LIN {X 0.031,Y -492.677,Z 365.442,A 0.000,B 0.000,C 90.000,E1 115.591} C_DIS
LIN {X -0.098,Y -489.173,Z 365.437,A 0.000,B 0.000,C 90.000,E1 114.695} C_DIS
LIN {X -0.238,Y -484.944,Z 365.431,A 0.000,B 0.000,C 90.000,E1 113.643} C_DIS
LIN {X 0.196,Y -479.146,Z 365.424,A 0.000,B 0.000,C 90.000,E1 112.206} C_DIS
LIN {X -0.106,Y -472.835,Z 365.416,A 0.000,B 0.000,C 90.000,E1 110.844} C_DIS
LIN {X -0.106,Y -464.087,Z 365.405,A 0.000,B 0.000,C 90.000,E1 108.960} C_DIS
LIN {X -0.172,Y -460.381,Z 365.401,A 0.000,B 0.000,C 90.000,E1 108.181} C_DIS
LIN {X -0.212,Y -460.379,Z 365.401,A 0.000,B 0.000,C 90.000,E1 108.181} C_DIS
LIN {X 0.188,Y -467.863,Z 365.383,A 0.000,B 0.000,C 90.000,E1 104.828} C_DIS
LIN {X -0.251,Y -475.421,Z 365.358,A 0.000,B 0.000,C 90.000,E1 100.489} C_DIS
LIN {X 0.054,Y -476.073,Z 365.356,A 0.000,B 0.000,C 90.000,E1 100.141} C_DIS
LIN {X -0.142,Y -481.996,Z 365.331,A 0.000,B 0.000,C 90.000,E1 95.511} C_DIS
LIN {X -0.161,Y -482.512,Z 365.325,A 0.000,B 0.000,C 90.000,E1 94.588} C_DIS
LIN {X 0.129,Y -485.445,Z 365.305,A 0.000,B 0.000,C 90.000,E1 90.859} C_DIS
LIN {X -0.219,Y -485.505,Z 365.301,A 0.000,B 0.000,C 90.000,E1 90.286} C_DIS
LIN {X 0.162,Y -486.380,Z 365.281,A 0.000,B 0.000,C 90.000,E1 86.560} C_DIS
LIN {X -0.014,Y -486.365,Z 365.279,A 0.000,B 0.000,C 90.000,E1 86.274} C_DIS
LIN {X 0.075,Y -484.690,Z 365.254,A 0.000,B 0.000,C 90.000,E1 81.659} C_DIS
LIN {X 0.220,Y -484.078,Z 365.250,A 0.000,B 0.000,C 90.000,E1 81.027} C_DIS
LIN {X -0.123,Y -480.642,Z 365.228,A 0.000,B 0.000,C 90.000,E1 77.061} C_DIS
LIN {X -0.158,Y -480.354,Z 365.226,A 0.000,B 0.000,C 90.000,E1 76.756} C_DIS
LIN {X -0.155,Y -475.588,Z 365.208,A 0.000,B 0.000,C 90.000,E1 73.433} C_DIS
LIN {X 0.260,Y -475.616,Z 365.208,A 0.000,B 0.000,C 90.000,E1 73.378} C_DIS
LIN {X 0.037,Y -482.998,Z 365.201,A 0.000,B 0.000,C 90.000,E1 72.236} C_DIS
LIN {X -0.116,Y -486.733,Z 365.198,A 0.000,B 0.000,C 90.000,E1 71.638} C_DIS
LIN {X -0.244,Y -490.378,Z 365.195,A 0.000,B 0.000,C 90.000,E1 71.040} C_DIS
LIN {X 0.028,Y -493.043,Z 365.192,A 0.000,B 0.000,C 90.000,E1 70.550} C_DIS
LIN {X -0.145,Y -495.741,Z 365.189,A 0.000,B 0.000,C 90.000,E1 70.115} C_DIS
LIN {X 0.049,Y -499.772,Z 365.185,A 0.000,B 0.000,C 90.000,E1 69.337} C_DIS
LIN {X -0.208,Y -504.048,Z 365.180,A 0.000,B 0.000,C 90.000,E1 68.465} C_DIS
LIN {X -0.037,Y -506.775,Z 365.177,A 0.000,B 0.000,C 90.000,E1 67.847} C_DIS
LIN {X -0.105,Y -511.591,Z 365.170,A 0.000,B 0.000,C 90.000,E1 66.666} C_DIS
LIN {X -0.233,Y -514.726,Z 365.165,A 0.000,B 0.000,C 90.000,E1 65.793} C_DIS
LIN {X -0.114,Y -517.640,Z 365.161,A 0.000,B 0.000,C 90.000,E1 64.897} C_DIS
LIN {X 0.151,Y -519.464,Z 365.157,A 0.000,B 0.000,C 90.000,E1 64.280} C_DIS
LIN {X -0.139,Y -522.117,Z 365.152,A 0.000,B 0.000,C 90.000,E1 63.435} C_DIS
LIN {X -0.160,Y -527.061,Z 365.143,A 0.000,B 0.000,C 90.000,E1 61.691} C_DIS
LIN {X -0.088,Y -531.857,Z 365.133,A 0.000,B 0.000,C 90.000,E1 59.950} C_DIS
LIN {X 0.001,Y -534.996,Z 365.127,A 0.000,B 0.000,C 90.000,E1 58.791} C_DIS
LIN {X -0.138,Y -538.016,Z 365.120,A 0.000,B 0.000,C 90.000,E1 57.661} C_DIS
LIN {X 0.085,Y -542.351,Z 365.111,A 0.000,B 0.000,C 90.000,E1 55.928} C_DIS
LIN {X -0.111,Y -545.003,Z 365.105,A 0.000,B 0.000,C 90.000,E1 54.815} C_DIS
LIN {X -0.317,Y -546.812,Z 365.100,A 0.000,B 0.000,C 90.000,E1 53.989} C_DIS
LIN {X -0.087,Y -549.488,Z 365.092,A 0.000,B 0.000,C 90.000,E1 52.557} C_DIS
LIN {X 0.073,Y -550.750,Z 365.087,A 0.000,B 0.000,C 90.000,E1 51.698} C_DIS
LIN {X -0.187,Y -551.579,Z 365.083,A 0.000,B 0.000,C 90.000,E1 50.884} C_DIS
LIN {X -0.083,Y -552.180,Z 365.078,A 0.000,B 0.000,C 90.000,E1 50.033} C_DIS
LIN {X 0.036,Y -552.398,Z 365.075,A 0.000,B 0.000,C 90.000,E1 49.461} C_DIS
LIN {X 0.156,Y -552.500,Z 365.070,A 0.000,B 0.000,C 90.000,E1 48.609} C_DIS
LIN {X -0.091,Y -552.312,Z 365.066,A 0.000,B 0.000,C 90.000,E1 47.796} C_DIS
LIN {X 0.025,Y -551.870,Z 365.061,A 0.000,B 0.000,C 90.000,E1 46.944} C_DIS
LIN {X -0.264,Y -551.137,Z 365.056,A 0.000,B 0.000,C 90.000,E1 46.134} C_DIS
LIN {X -0.135,Y -549.862,Z 365.050,A 0.000,B 0.000,C 90.000,E1 45.000} C_DIS
LIN {X 0.007,Y -548.109,Z 365.042,A 0.000,B 0.000,C 90.000,E1 43.581} C_DIS
LIN {X 0.142,Y -545.398,Z 365.031,A 0.000,B 0.000,C 90.000,E1 41.595} C_DIS
LIN {X -0.145,Y -543.179,Z 365.022,A 0.000,B 0.000,C 90.000,E1 39.930} C_DIS
LIN {X -0.045,Y -540.492,Z 365.011,A 0.000,B 0.000,C 90.000,E1 37.935} C_DIS
LIN {X 0.066,Y -538.243,Z 365.001,A 0.000,B 0.000,C 90.000,E1 36.217} C_DIS
LIN {X -0.188,Y -535.980,Z 364.992,A 0.000,B 0.000,C 90.000,E1 34.532} C_DIS
LIN {X -0.052,Y -533.823,Z 364.982,A 0.000,B 0.000,C 90.000,E1 32.801} C_DIS
LIN {X 0.215,Y -532.034,Z 364.974,A 0.000,B 0.000,C 90.000,E1 31.337} C_DIS
LIN {X 0.160,Y -530.007,Z 364.965,A 0.000,B 0.000,C 90.000,E1 29.617} C_DIS
LIN {X -0.247,Y -527.759,Z 364.953,A 0.000,B 0.000,C 90.000,E1 27.641} C_DIS
LIN {X -0.028,Y -525.601,Z 364.942,A 0.000,B 0.000,C 90.000,E1 25.591} C_DIS
LIN {X 0.221,Y -523.874,Z 364.933,A 0.000,B 0.000,C 90.000,E1 23.823} C_DIS
LIN {X 0.061,Y -522.555,Z 364.924,A 0.000,B 0.000,C 90.000,E1 22.386} C_DIS
LIN {X -0.048,Y -520.702,Z 364.911,A 0.000,B 0.000,C 90.000,E1 20.066} C_DIS
LIN {X 0.144,Y -519.352,Z 364.900,A 0.000,B 0.000,C 90.000,E1 18.000} C_DIS
LIN {X -0.114,Y -518.754,Z 364.894,A 0.000,B 0.000,C 90.000,E1 16.858} C_DIS
LIN {X 0.207,Y -517.916,Z 364.882,A 0.000,B 0.000,C 90.000,E1 14.773} C_DIS
LIN {X -0.176,Y -517.362,Z 364.866,A 0.000,B 0.000,C 90.000,E1 11.883} C_DIS
LIN {X 0.149,Y -517.388,Z 364.853,A 0.000,B 0.000,C 90.000,E1 9.500} C_DIS
LIN {X 0.125,Y -517.389,Z 364.850,A 0.000,B 0.000,C 90.000,E1 8.916} C_DIS
LIN {X 0.007,Y -517.728,Z 364.845,A 0.000,B 0.000,C 90.000,E1 8.049} C_DIS
LIN {X -0.060,Y -519.631,Z 364.822,A 0.000,B 0.000,C 90.000,E1 3.955} C_DIS
LIN {X -0.082,Y -522.363,Z 364.804,A 0.000,B 0.000,C 90.000,E1 0.745} C_DIS
LIN {X -0.091,Y -526.446,Z 364.786,A 0.000,B 0.000,C 90.000,E1 357.478} C_DIS
LIN {X -0.247,Y -529.588,Z 364.775,A 0.000,B 0.000,C 90.000,E1 355.469} C_DIS
LIN {X -0.228,Y -533.117,Z 364.764,A 0.000,B 0.000,C 90.000,E1 353.451} C_DIS
LIN {X -0.116,Y -537.025,Z 364.752,A 0.000,B 0.000,C 90.000,E1 351.432} C_DIS
LIN {X 0.126,Y -545.013,Z 364.733,A 0.000,B 0.000,C 90.000,E1 347.993} C_DIS
LIN {X -0.031,Y -551.141,Z 364.721,A 0.000,B 0.000,C 90.000,E1 345.755} C_DIS
LIN {X 0.001,Y -556.922,Z 364.710,A 0.000,B 0.000,C 90.000,E1 343.795} C_DIS
LIN {X -0.106,Y -561.147,Z 364.702,A 0.000,B 0.000,C 90.000,E1 342.417} C_DIS
LIN {X 0.178,Y -566.255,Z 364.693,A 0.000,B 0.000,C 90.000,E1 340.732} C_DIS
LIN {X -0.126,Y -570.563,Z 364.685,A 0.000,B 0.000,C 90.000,E1 339.390} C_DIS
LIN {X 0.217,Y -575.641,Z 364.676,A 0.000,B 0.000,C 90.000,E1 337.720} C_DIS
LIN {X 0.286,Y -579.970,Z 364.669,A 0.000,B 0.000,C 90.000,E1 336.357} C_DIS
LIN {X 0.160,Y -586.014,Z 364.658,A 0.000,B 0.000,C 90.000,E1 334.485} C_DIS
LIN {X 0.052,Y -593.076,Z 364.647,A 0.000,B 0.000,C 90.000,E1 332.359} C_DIS
LIN {X -0.047,Y -596.678,Z 364.641,A 0.000,B 0.000,C 90.000,E1 331.307} C_DIS
LIN {X -0.093,Y -600.308,Z 364.635,A 0.000,B 0.000,C 90.000,E1 330.255} C_DIS
LIN {X 0.083,Y -605.802,Z 364.626,A 0.000,B 0.000,C 90.000,E1 328.663} C_DIS
LIN {X -0.157,Y -611.211,Z 364.617,A 0.000,B 0.000,C 90.000,E1 327.120} C_DIS
LIN {X -0.170,Y -617.620,Z 364.607,A 0.000,B 0.000,C 90.000,E1 325.308} C_DIS
LIN {X -0.028,Y -624.176,Z 364.597,A 0.000,B 0.000,C 90.000,E1 323.497} C_DIS
LIN {X 0.306,Y -628.949,Z 364.590,A 0.000,B 0.000,C 90.000,E1 322.190} C_DIS
LIN {X 0.350,Y -637.363,Z 364.577,A 0.000,B 0.000,C 90.000,E1 319.908} C_DIS
LIN {X 0.021,Y -641.197,Z 364.572,A 0.000,B 0.000,C 90.000,E1 318.933} C_DIS
LIN {X 0.090,Y -645.615,Z 364.565,A 0.000,B 0.000,C 90.000,E1 317.676} C_DIS
LIN {X 0.050,Y -653.617,Z 364.553,A 0.000,B 0.000,C 90.000,E1 315.445} C_DIS
LIN {X 0.291,Y -658.944,Z 364.544,A 0.000,B 0.000,C 90.000,E1 313.947} C_DIS
LIN {X -0.290,Y -664.100,Z 364.536,A 0.000,B 0.000,C 90.000,E1 312.528} C_DIS
LIN {X 0.164,Y -667.540,Z 364.531,A 0.000,B 0.000,C 90.000,E1 311.515} C_DIS
LIN {X -0.210,Y -671.484,Z 364.524,A 0.000,B 0.000,C 90.000,E1 310.334} C_DIS
LIN {X -0.085,Y -675.435,Z 364.517,A 0.000,B 0.000,C 90.000,E1 309.116} C_DIS
LIN {X -0.350,Y -678.537,Z 364.512,A 0.000,B 0.000,C 90.000,E1 308.177} C_DIS
LIN {X 0.382,Y -681.266,Z 364.507,A 0.000,B 0.000,C 90.000,E1 307.156} C_DIS
LIN {X 0.191,Y -683.841,Z 364.501,A 0.000,B 0.000,C 90.000,E1 306.217} C_DIS
LIN {X -0.372,Y -686.227,Z 364.496,A 0.000,B 0.000,C 90.000,E1 305.311} C_DIS
LIN {X 0.050,Y -688.341,Z 364.491,A 0.000,B 0.000,C 90.000,E1 304.326} C_DIS
LIN {X -0.097,Y -689.746,Z 364.487,A 0.000,B 0.000,C 90.000,E1 303.627} C_DIS
LIN {X 0.344,Y -690.890,Z 364.483,A 0.000,B 0.000,C 90.000,E1 302.880} C_DIS
LIN {X 0.074,Y -692.274,Z 364.478,A 0.000,B 0.000,C 90.000,E1 301.957} C_DIS
LIN {X 0.312,Y -692.953,Z 364.475,A 0.000,B 0.000,C 90.000,E1 301.465} C_DIS
LIN {X -0.165,Y -693.622,Z 364.471,A 0.000,B 0.000,C 90.000,E1 300.797} C_DIS
LIN {X -0.280,Y -693.986,Z 364.468,A 0.000,B 0.000,C 90.000,E1 300.335} C_DIS
LIN {X 0.101,Y -694.209,Z 364.463,A 0.000,B 0.000,C 90.000,E1 299.361} C_DIS
LIN {X -0.006,Y -694.162,Z 364.461,A 0.000,B 0.000,C 90.000,E1 298.899} C_DIS
LIN {X 0.134,Y -693.618,Z 364.457,A 0.000,B 0.000,C 90.000,E1 298.180} C_DIS
LIN {X 0.145,Y -692.090,Z 364.450,A 0.000,B 0.000,C 90.000,E1 297.001} C_DIS
LIN {X 0.189,Y -690.657,Z 364.445,A 0.000,B 0.000,C 90.000,E1 296.052} C_DIS
LIN {X 0.280,Y -689.460,Z 364.441,A 0.000,B 0.000,C 90.000,E1 295.335} C_DIS
LIN {X 0.288,Y -687.540,Z 364.436,A 0.000,B 0.000,C 90.000,E1 294.387} C_DIS
LIN {X 0.213,Y -684.989,Z 364.429,A 0.000,B 0.000,C 90.000,E1 293.206} C_DIS
LIN {X -0.103,Y -682.772,Z 364.424,A 0.000,B 0.000,C 90.000,E1 292.280} C_DIS
LIN {X -0.064,Y -679.228,Z 364.416,A 0.000,B 0.000,C 90.000,E1 290.844} C_DIS
LIN {X 0.055,Y -675.760,Z 364.408,A 0.000,B 0.000,C 90.000,E1 289.396} C_DIS
LIN {X 0.249,Y -673.445,Z 364.402,A 0.000,B 0.000,C 90.000,E1 288.417} C_DIS
LIN {X 0.112,Y -668.889,Z 364.392,A 0.000,B 0.000,C 90.000,E1 286.496} C_DIS
LIN {X 0.147,Y -663.586,Z 364.378,A 0.000,B 0.000,C 90.000,E1 284.064} C_DIS
LIN {X 0.152,Y -658.265,Z 364.362,A 0.000,B 0.000,C 90.000,E1 281.130} C_DIS
LIN {X 0.060,Y -654.842,Z 364.348,A 0.000,B 0.000,C 90.000,E1 278.681} C_DIS
LIN {X -0.150,Y -651.967,Z 364.332,A 0.000,B 0.000,C 90.000,E1 275.739} C_DIS
LIN {X 0.288,Y -650.524,Z 364.317,A 0.000,B 0.000,C 90.000,E1 272.980} C_DIS
LIN {X -0.294,Y -649.937,Z 364.304,A 0.000,B 0.000,C 90.000,E1 270.802} C_DIS
LIN {X 0.015,Y -650.410,Z 364.285,A 0.000,B 0.000,C 90.000,E1 267.306} C_DIS
LIN {X 0.112,Y -651.031,Z 364.277,A 0.000,B 0.000,C 90.000,E1 265.812} C_DIS
LIN {X 0.007,Y -651.804,Z 364.267,A 0.000,B 0.000,C 90.000,E1 264.090} C_DIS
LIN {X -0.180,Y -652.598,Z 364.256,A 0.000,B 0.000,C 90.000,E1 262.129} C_DIS
LIN {X -0.039,Y -652.961,Z 364.252,A 0.000,B 0.000,C 90.000,E1 261.376} C_DIS
LIN {X 0.105,Y -652.989,Z 364.248,A 0.000,B 0.000,C 90.000,E1 260.622} C_DIS
LIN {X -0.134,Y -652.869,Z 364.240,A 0.000,B 0.000,C 90.000,E1 259.162} C_DIS
LIN {X 0.268,Y -652.672,Z 364.232,A 0.000,B 0.000,C 90.000,E1 257.645} C_DIS
LIN {X -0.101,Y -652.414,Z 364.227,A 0.000,B 0.000,C 90.000,E1 256.937} C_DIS
LIN {X -0.085,Y -651.414,Z 364.221,A 0.000,B 0.000,C 90.000,E1 255.700} C_DIS
LIN {X 0.165,Y -650.736,Z 364.216,A 0.000,B 0.000,C 90.000,E1 254.936} C_DIS
LIN {X -0.050,Y -649.669,Z 364.212,A 0.000,B 0.000,C 90.000,E1 254.212} C_DIS
LIN {X 0.172,Y -648.378,Z 364.208,A 0.000,B 0.000,C 90.000,E1 253.449} C_DIS
LIN {X 0.083,Y -647.443,Z 364.205,A 0.000,B 0.000,C 90.000,E1 252.960} C_DIS
LIN {X -0.150,Y -645.773,Z 364.201,A 0.000,B 0.000,C 90.000,E1 252.236} C_DIS
LIN {X 0.214,Y -643.871,Z 364.197,A 0.000,B 0.000,C 90.000,E1 251.456} C_DIS
LIN {X 0.107,Y -642.470,Z 364.194,A 0.000,B 0.000,C 90.000,E1 250.967} C_DIS
LIN {X -0.345,Y -639.212,Z 364.189,A 0.000,B 0.000,C 90.000,E1 250.007} C_DIS
LIN {X 0.197,Y -635.669,Z 364.183,A 0.000,B 0.000,C 90.000,E1 248.954} C_DIS
LIN {X -0.128,Y -631.902,Z 364.178,A 0.000,B 0.000,C 90.000,E1 247.975} C_DIS
LIN {X 0.335,Y -626.967,Z 364.171,A 0.000,B 0.000,C 90.000,E1 246.666} C_DIS
LIN {X 0.140,Y -621.804,Z 364.164,A 0.000,B 0.000,C 90.000,E1 245.409} C_DIS
LIN {X -0.156,Y -615.473,Z 364.155,A 0.000,B 0.000,C 90.000,E1 243.896} C_DIS
LIN {X -0.352,Y -608.026,Z 364.145,A 0.000,B 0.000,C 90.000,E1 242.103} C_DIS
LIN {X -0.084,Y -601.654,Z 364.136,A 0.000,B 0.000,C 90.000,E1 240.511} C_DIS
LIN {X 0.063,Y -595.379,Z 364.127,A 0.000,B 0.000,C 90.000,E1 238.918} C_DIS
LIN {X -0.290,Y -585.515,Z 364.113,A 0.000,B 0.000,C 90.000,E1 236.294} C_DIS
LIN {X 0.159,Y -577.276,Z 364.099,A 0.000,B 0.000,C 90.000,E1 233.829} C_DIS
LIN {X 0.126,Y -572.773,Z 364.092,A 0.000,B 0.000,C 90.000,E1 232.477} C_DIS
LIN {X -0.316,Y -566.944,Z 364.083,A 0.000,B 0.000,C 90.000,E1 230.884} C_DIS
LIN {X 0.059,Y -558.457,Z 364.069,A 0.000,B 0.000,C 90.000,E1 228.366} C_DIS
LIN {X 0.317,Y -554.841,Z 364.063,A 0.000,B 0.000,C 90.000,E1 227.229} C_DIS
LIN {X -0.243,Y -550.314,Z 364.055,A 0.000,B 0.000,C 90.000,E1 225.891} C_DIS
LIN {X -0.130,Y -546.711,Z 364.049,A 0.000,B 0.000,C 90.000,E1 224.757} C_DIS
LIN {X -0.052,Y -540.419,Z 364.038,A 0.000,B 0.000,C 90.000,E1 222.771} C_DIS
LIN {X -0.098,Y -536.030,Z 364.030,A 0.000,B 0.000,C 90.000,E1 221.353} C_DIS
LIN {X -0.202,Y -529.943,Z 364.019,A 0.000,B 0.000,C 90.000,E1 219.358} C_DIS
LIN {X -0.002,Y -524.922,Z 364.009,A 0.000,B 0.000,C 90.000,E1 217.604} C_DIS
LIN {X -0.280,Y -519.322,Z 363.998,A 0.000,B 0.000,C 90.000,E1 215.598} C_DIS
LIN {X 0.135,Y -513.916,Z 363.986,A 0.000,B 0.000,C 90.000,E1 213.499} C_DIS
LIN {X -0.160,Y -508.947,Z 363.975,A 0.000,B 0.000,C 90.000,E1 211.465} C_DIS
LIN {X 0.285,Y -504.162,Z 363.963,A 0.000,B 0.000,C 90.000,E1 209.333} C_DIS
LIN {X 0.111,Y -499.534,Z 363.952,A 0.000,B 0.000,C 90.000,E1 207.257} C_DIS
LIN {X -0.061,Y -496.198,Z 363.943,A 0.000,B 0.000,C 90.000,E1 205.771} C_DIS
LIN {X 0.016,Y -491.422,Z 363.931,A 0.000,B 0.000,C 90.000,E1 203.643} C_DIS
LIN {X -0.267,Y -487.865,Z 363.923,A 0.000,B 0.000,C 90.000,E1 202.153} C_DIS
LIN {X -0.153,Y -483.540,Z 363.913,A 0.000,B 0.000,C 90.000,E1 200.301} C_DIS
LIN {X -0.023,Y -478.616,Z 363.901,A 0.000,B 0.000,C 90.000,E1 198.127} C_DIS
LIN {X 0.042,Y -475.354,Z 363.892,A 0.000,B 0.000,C 90.000,E1 196.567} C_DIS
LIN {X 0.038,Y -472.146,Z 363.883,A 0.000,B 0.000,C 90.000,E1 195.009} C_DIS
LIN {X -0.255,Y -467.280,Z 363.870,A 0.000,B 0.000,C 90.000,E1 192.535} C_DIS
LIN {X -0.136,Y -463.231,Z 363.857,A 0.000,B 0.000,C 90.000,E1 190.310} C_DIS
LIN {X 0.132,Y -460.521,Z 363.848,A 0.000,B 0.000,C 90.000,E1 188.690} C_DIS
LIN {X -0.160,Y -455.953,Z 363.832,A 0.000,B 0.000,C 90.000,E1 185.853} C_DIS
LIN {X 0.071,Y -453.224,Z 363.822,A 0.000,B 0.000,C 90.000,E1 183.898} C_DIS
LIN {X -0.060,Y -449.522,Z 363.804,A 0.000,B 0.000,C 90.000,E1 180.688} C_DIS
LIN {X -0.169,Y -447.293,Z 363.789,A 0.000,B 0.000,C 90.000,E1 178.108} C_DIS
LIN {X -0.156,Y -445.691,Z 363.773,A 0.000,B 0.000,C 90.000,E1 175.179} C_DIS
LIN {X -0.048,Y -444.869,Z 363.751,A 0.000,B 0.000,C 90.000,E1 171.254} C_DIS
LIN {X -0.051,Y -445.454,Z 363.733,A 0.000,B 0.000,C 90.000,E1 167.993} C_DIS
LIN {X -0.014,Y -448.174,Z 363.708,A 0.000,B 0.000,C 90.000,E1 163.433} C_DIS
LIN {X 0.101,Y -452.644,Z 363.685,A 0.000,B 0.000,C 90.000,E1 159.209} C_DIS
LIN {X 0.075,Y -458.323,Z 363.663,A 0.000,B 0.000,C 90.000,E1 155.357} C_DIS
LIN {X -0.133,Y -465.675,Z 363.642,A 0.000,B 0.000,C 90.000,E1 151.563} C_DIS
LIN {X -0.121,Y -474.840,Z 363.621,A 0.000,B 0.000,C 90.000,E1 147.788} C_DIS
LIN {X -0.155,Y -484.184,Z 363.604,A 0.000,B 0.000,C 90.000,E1 144.689} C_DIS
LIN {X 0.095,Y -493.378,Z 363.588,A 0.000,B 0.000,C 90.000,E1 141.904} C_DIS
LIN {X -0.319,Y -498.448,Z 363.580,A 0.000,B 0.000,C 90.000,E1 140.436} C_DIS
LIN {X -0.324,Y -503.318,Z 363.572,A 0.000,B 0.000,C 90.000,E1 138.933} C_DIS
LIN {X -0.133,Y -507.101,Z 363.565,A 0.000,B 0.000,C 90.000,E1 137.715} C_DIS
LIN {X -0.016,Y -511.352,Z 363.557,A 0.000,B 0.000,C 90.000,E1 136.215} C_DIS
LIN {X -0.187,Y -515.020,Z 363.549,A 0.000,B 0.000,C 90.000,E1 134.757} C_DIS
LIN {X -0.113,Y -516.934,Z 363.544,A 0.000,B 0.000,C 90.000,E1 133.866} C_DIS
LIN {X -0.021,Y -518.432,Z 363.539,A 0.000,B 0.000,C 90.000,E1 132.975} C_DIS
LIN {X 0.116,Y -519.688,Z 363.534,A 0.000,B 0.000,C 90.000,E1 132.081} C_DIS
LIN {X 0.169,Y -520.890,Z 363.527,A 0.000,B 0.000,C 90.000,E1 130.906} C_DIS
LIN {X -0.111,Y -521.448,Z 363.521,A 0.000,B 0.000,C 90.000,E1 129.769} C_DIS
LIN {X 0.014,Y -521.274,Z 363.514,A 0.000,B 0.000,C 90.000,E1 128.588} C_DIS
LIN {X -0.135,Y -520.680,Z 363.510,A 0.000,B 0.000,C 90.000,E1 127.729} C_DIS
LIN {X 0.080,Y -519.437,Z 363.503,A 0.000,B 0.000,C 90.000,E1 126.537} C_DIS
LIN {X -0.137,Y -518.012,Z 363.497,A 0.000,B 0.000,C 90.000,E1 125.391} C_DIS
LIN {X 0.107,Y -516.681,Z 363.492,A 0.000,B 0.000,C 90.000,E1 124.485} C_DIS
LIN {X -0.097,Y -515.121,Z 363.487,A 0.000,B 0.000,C 90.000,E1 123.627} C_DIS
LIN {X 0.177,Y -512.762,Z 363.480,A 0.000,B 0.000,C 90.000,E1 122.418} C_DIS
LIN {X 0.079,Y -510.809,Z 363.475,A 0.000,B 0.000,C 90.000,E1 121.544} C_DIS
LIN {X -0.146,Y -507.845,Z 363.469,A 0.000,B 0.000,C 90.000,E1 120.384} C_DIS
LIN {X -0.236,Y -504.662,Z 363.462,A 0.000,B 0.000,C 90.000,E1 119.205} C_DIS
LIN {X 0.007,Y -502.020,Z 363.457,A 0.000,B 0.000,C 90.000,E1 118.281} C_DIS
LIN {X -0.122,Y -497.242,Z 363.449,A 0.000,B 0.000,C 90.000,E1 116.796} C_DIS
LIN {X -0.154,Y -493.197,Z 363.442,A 0.000,B 0.000,C 90.000,E1 115.591} C_DIS
LIN {X 0.169,Y -489.810,Z 363.437,A 0.000,B 0.000,C 90.000,E1 114.643} C_DIS
LIN {X 0.251,Y -484.504,Z 363.429,A 0.000,B 0.000,C 90.000,E1 113.259} C_DIS
LIN {X -0.176,Y -479.493,Z 363.423,A 0.000,B 0.000,C 90.000,E1 112.078} C_DIS
LIN {X 0.180,Y -472.559,Z 363.414,A 0.000,B 0.000,C 90.000,E1 110.482} C_DIS
LIN {X -0.015,Y -464.652,Z 363.404,A 0.000,B 0.000,C 90.000,E1 108.779} C_DIS
LIN {X 0.042,Y -460.806,Z 363.400,A 0.000,B 0.000,C 90.000,E1 107.946} C_DIS
LIN {X 0.002,Y -460.802,Z 363.400,A 0.000,B 0.000,C 90.000,E1 107.946} C_DIS
LIN {X 0.151,Y -467.595,Z 363.383,A 0.000,B 0.000,C 90.000,E1 104.954} C_DIS
LIN {X -0.118,Y -468.593,Z 363.380,A 0.000,B 0.000,C 90.000,E1 104.356} C_DIS
LIN {X 0.109,Y -475.822,Z 363.357,A 0.000,B 0.000,C 90.000,E1 100.254} C_DIS
LIN {X -0.053,Y -476.315,Z 363.355,A 0.000,B 0.000,C 90.000,E1 99.962} C_DIS
LIN {X -0.106,Y -481.806,Z 363.331,A 0.000,B 0.000,C 90.000,E1 95.625} C_DIS
LIN {X 0.221,Y -482.175,Z 363.330,A 0.000,B 0.000,C 90.000,E1 95.277} C_DIS
LIN {X 0.156,Y -485.319,Z 363.306,A 0.000,B 0.000,C 90.000,E1 90.974} C_DIS
LIN {X -0.020,Y -485.536,Z 363.304,A 0.000,B 0.000,C 90.000,E1 90.688} C_DIS
LIN {X 0.187,Y -486.324,Z 363.282,A 0.000,B 0.000,C 90.000,E1 86.674} C_DIS
LIN {X -0.163,Y -486.298,Z 363.278,A 0.000,B 0.000,C 90.000,E1 86.102} C_DIS
LIN {X 0.041,Y -484.695,Z 363.254,A 0.000,B 0.000,C 90.000,E1 81.781} C_DIS
LIN {X -0.090,Y -484.588,Z 363.253,A 0.000,B 0.000,C 90.000,E1 81.489} C_DIS
LIN {X -0.210,Y -480.524,Z 363.227,A 0.000,B 0.000,C 90.000,E1 76.881} C_DIS
LIN {X 0.110,Y -475.776,Z 363.209,A 0.000,B 0.000,C 90.000,E1 73.559} C_DIS
LIN {X 0.069,Y -475.794,Z 363.209,A 0.000,B 0.000,C 90.000,E1 73.559} C_DIS
LIN {X -0.007,Y -481.372,Z 363.204,A 0.000,B 0.000,C 90.000,E1 72.670} C_DIS
LIN {X -0.173,Y -486.947,Z 363.199,A 0.000,B 0.000,C 90.000,E1 71.764} C_DIS
LIN {X 0.101,Y -491.337,Z 363.194,A 0.000,B 0.000,C 90.000,E1 70.967} C_DIS
LIN {X -0.205,Y -495.585,Z 363.190,A 0.000,B 0.000,C 90.000,E1 70.242} C_DIS
LIN {X 0.162,Y -499.452,Z 363.186,A 0.000,B 0.000,C 90.000,E1 69.444} C_DIS
LIN {X -0.079,Y -502.844,Z 363.182,A 0.000,B 0.000,C 90.000,E1 68.720} C_DIS
LIN {X 0.193,Y -503.597,Z 363.181,A 0.000,B 0.000,C 90.000,E1 68.539} C_DIS
LIN {X 0.081,Y -505.422,Z 363.178,A 0.000,B 0.000,C 90.000,E1 68.103} C_DIS
LIN {X -0.112,Y -506.116,Z 363.178,A 0.000,B 0.000,C 90.000,E1 67.975} C_DIS
LIN {X -0.196,Y -510.811,Z 363.171,A 0.000,B 0.000,C 90.000,E1 66.794} C_DIS
LIN {X 0.022,Y -512.978,Z 363.168,A 0.000,B 0.000,C 90.000,E1 66.177} C_DIS
LIN {X 0.119,Y -515.973,Z 363.163,A 0.000,B 0.000,C 90.000,E1 65.281} C_DIS
LIN {X 0.034,Y -518.711,Z 363.158,A 0.000,B 0.000,C 90.000,E1 64.409} C_DIS
LIN {X -0.124,Y -522.149,Z 363.151,A 0.000,B 0.000,C 90.000,E1 63.256} C_DIS
LIN {X -0.154,Y -527.053,Z 363.142,A 0.000,B 0.000,C 90.000,E1 61.513} C_DIS
LIN {X 0.145,Y -532.604,Z 363.130,A 0.000,B 0.000,C 90.000,E1 59.459} C_DIS
LIN {X -0.033,Y -536.524,Z 363.122,A 0.000,B 0.000,C 90.000,E1 58.043} C_DIS
LIN {X 0.335,Y -541.669,Z 363.111,A 0.000,B 0.000,C 90.000,E1 56.008} C_DIS
LIN {X 0.160,Y -545.001,Z 363.104,A 0.000,B 0.000,C 90.000,E1 54.609} C_DIS
LIN {X -0.047,Y -546.822,Z 363.099,A 0.000,B 0.000,C 90.000,E1 53.783} C_DIS
LIN {X 0.182,Y -549.536,Z 363.091,A 0.000,B 0.000,C 90.000,E1 52.351} C_DIS
LIN {X -0.146,Y -550.425,Z 363.088,A 0.000,B 0.000,C 90.000,E1 51.823} C_DIS
LIN {X 0.079,Y -551.730,Z 363.082,A 0.000,B 0.000,C 90.000,E1 50.678} C_DIS
LIN {X 0.184,Y -552.378,Z 363.077,A 0.000,B 0.000,C 90.000,E1 49.828} C_DIS
LIN {X -0.002,Y -552.832,Z 363.071,A 0.000,B 0.000,C 90.000,E1 48.728} C_DIS
LIN {X 0.118,Y -552.830,Z 363.066,A 0.000,B 0.000,C 90.000,E1 47.877} C_DIS
LIN {X -0.165,Y -552.506,Z 363.061,A 0.000,B 0.000,C 90.000,E1 47.067} C_DIS
LIN {X -0.044,Y -551.978,Z 363.057,A 0.000,B 0.000,C 90.000,E1 46.215} C_DIS
LIN {X 0.096,Y -550.856,Z 363.051,A 0.000,B 0.000,C 90.000,E1 45.081} C_DIS
LIN {X -0.141,Y -549.168,Z 363.043,A 0.000,B 0.000,C 90.000,E1 43.704} C_DIS
LIN {X 0.054,Y -546.458,Z 363.032,A 0.000,B 0.000,C 90.000,E1 41.714} C_DIS
LIN {X 0.153,Y -544.243,Z 363.022,A 0.000,B 0.000,C 90.000,E1 40.011} C_DIS
LIN {X 0.281,Y -541.547,Z 363.011,A 0.000,B 0.000,C 90.000,E1 38.016} C_DIS
LIN {X -0.018,Y -539.283,Z 363.002,A 0.000,B 0.000,C 90.000,E1 36.343} C_DIS
LIN {X 0.187,Y -537.049,Z 362.992,A 0.000,B 0.000,C 90.000,E1 34.612} C_DIS
LIN {X 0.060,Y -534.894,Z 362.983,A 0.000,B 0.000,C 90.000,E1 32.911} C_DIS
LIN {X 0.185,Y -533.119,Z 362.975,A 0.000,B 0.000,C 90.000,E1 31.465} C_DIS
LIN {X 0.151,Y -531.130,Z 362.965,A 0.000,B 0.000,C 90.000,E1 29.745} C_DIS
LIN {X -0.230,Y -528.866,Z 362.954,A 0.000,B 0.000,C 90.000,E1 27.769} C_DIS
LIN {X -0.151,Y -526.972,Z 362.945,A 0.000,B 0.000,C 90.000,E1 26.027} C_DIS
LIN {X 0.293,Y -525.010,Z 362.933,A 0.000,B 0.000,C 90.000,E1 23.951} C_DIS
LIN {X 0.316,Y -523.395,Z 362.924,A 0.000,B 0.000,C 90.000,E1 22.206} C_DIS
LIN {X -0.255,Y -521.587,Z 362.911,A 0.000,B 0.000,C 90.000,E1 19.939} C_DIS
LIN {X -0.044,Y -520.274,Z 362.899,A 0.000,B 0.000,C 90.000,E1 17.873} C_DIS
LIN {X -0.174,Y -519.444,Z 362.890,A 0.000,B 0.000,C 90.000,E1 16.134} C_DIS
LIN {X 0.035,Y -518.798,Z 362.880,A 0.000,B 0.000,C 90.000,E1 14.356} C_DIS
LIN {X 0.094,Y -518.430,Z 362.867,A 0.000,B 0.000,C 90.000,E1 12.007} C_DIS
LIN {X 0.038,Y -518.500,Z 362.854,A 0.000,B 0.000,C 90.000,E1 9.670} C_DIS
LIN {X -0.071,Y -518.582,Z 362.849,A 0.000,B 0.000,C 90.000,E1 8.803} C_DIS
LIN {X -0.182,Y -518.960,Z 362.842,A 0.000,B 0.000,C 90.000,E1 7.644} C_DIS
LIN {X -0.172,Y -520.861,Z 362.821,A 0.000,B 0.000,C 90.000,E1 3.841} C_DIS
LIN {X -0.142,Y -523.668,Z 362.803,A 0.000,B 0.000,C 90.000,E1 0.630} C_DIS
LIN {X -0.026,Y -527.212,Z 362.788,A 0.000,B 0.000,C 90.000,E1 357.764} C_DIS
LIN {X -0.156,Y -530.324,Z 362.776,A 0.000,B 0.000,C 90.000,E1 355.755} C_DIS
LIN {X -0.204,Y -533.309,Z 362.767,A 0.000,B 0.000,C 90.000,E1 354.033} C_DIS
LIN {X -0.046,Y -537.669,Z 362.754,A 0.000,B 0.000,C 90.000,E1 351.724} C_DIS
LIN {X 0.219,Y -545.491,Z 362.735,A 0.000,B 0.000,C 90.000,E1 348.285} C_DIS
LIN {X -0.053,Y -551.571,Z 362.723,A 0.000,B 0.000,C 90.000,E1 346.061} C_DIS
LIN {X -0.025,Y -557.286,Z 362.712,A 0.000,B 0.000,C 90.000,E1 344.102} C_DIS
LIN {X -0.132,Y -561.551,Z 362.704,A 0.000,B 0.000,C 90.000,E1 342.725} C_DIS
LIN {X -0.051,Y -567.501,Z 362.693,A 0.000,B 0.000,C 90.000,E1 340.786} C_DIS
LIN {X 0.205,Y -571.814,Z 362.686,A 0.000,B 0.000,C 90.000,E1 339.390} C_DIS
LIN {X 0.201,Y -577.774,Z 362.675,A 0.000,B 0.000,C 90.000,E1 337.486} C_DIS
LIN {X -0.234,Y -582.123,Z 362.668,A 0.000,B 0.000,C 90.000,E1 336.177} C_DIS
LIN {X 0.052,Y -587.345,Z 362.659,A 0.000,B 0.000,C 90.000,E1 334.537} C_DIS
LIN {X 0.086,Y -593.551,Z 362.648,A 0.000,B 0.000,C 90.000,E1 332.666} C_DIS
LIN {X -0.373,Y -598.064,Z 362.641,A 0.000,B 0.000,C 90.000,E1 331.385} C_DIS
LIN {X -0.322,Y -604.429,Z 362.631,A 0.000,B 0.000,C 90.000,E1 329.537} C_DIS
LIN {X 0.045,Y -608.104,Z 362.625,A 0.000,B 0.000,C 90.000,E1 328.456} C_DIS
LIN {X -0.148,Y -613.513,Z 362.616,A 0.000,B 0.000,C 90.000,E1 326.914} C_DIS
LIN {X 0.094,Y -619.077,Z 362.608,A 0.000,B 0.000,C 90.000,E1 325.341} C_DIS
LIN {X -0.212,Y -624.643,Z 362.599,A 0.000,B 0.000,C 90.000,E1 323.829} C_DIS
LIN {X -0.247,Y -629.281,Z 362.592,A 0.000,B 0.000,C 90.000,E1 322.557} C_DIS
LIN {X -0.193,Y -632.932,Z 362.586,A 0.000,B 0.000,C 90.000,E1 321.537} C_DIS
LIN {X -0.018,Y -640.417,Z 362.575,A 0.000,B 0.000,C 90.000,E1 319.504} C_DIS
LIN {X -0.223,Y -643.176,Z 362.571,A 0.000,B 0.000,C 90.000,E1 318.771} C_DIS
LIN {X 0.358,Y -647.451,Z 362.564,A 0.000,B 0.000,C 90.000,E1 317.472} C_DIS
LIN {X -0.063,Y -654.544,Z 362.553,A 0.000,B 0.000,C 90.000,E1 315.526} C_DIS
LIN {X 0.194,Y -659.780,Z 362.545,A 0.000,B 0.000,C 90.000,E1 314.028} C_DIS
LIN {X -0.358,Y -664.049,Z 362.538,A 0.000,B 0.000,C 90.000,E1 312.852} C_DIS
LIN {X 0.098,Y -667.523,Z 362.533,A 0.000,B 0.000,C 90.000,E1 311.838} C_DIS
LIN {X 0.164,Y -671.479,Z 362.526,A 0.000,B 0.000,C 90.000,E1 310.620} C_DIS
LIN {X -0.140,Y -675.445,Z 362.519,A 0.000,B 0.000,C 90.000,E1 309.439} C_DIS
LIN {X 0.039,Y -679.273,Z 362.512,A 0.000,B 0.000,C 90.000,E1 308.222} C_DIS
LIN {X -0.180,Y -682.018,Z 362.507,A 0.000,B 0.000,C 90.000,E1 307.282} C_DIS
LIN {X -0.197,Y -685.179,Z 362.500,A 0.000,B 0.000,C 90.000,E1 306.091} C_DIS
LIN {X 0.216,Y -687.439,Z 362.495,A 0.000,B 0.000,C 90.000,E1 305.105} C_DIS
LIN {X 0.066,Y -688.957,Z 362.491,A 0.000,B 0.000,C 90.000,E1 304.405} C_DIS
LIN {X 0.292,Y -689.921,Z 362.489,A 0.000,B 0.000,C 90.000,E1 303.913} C_DIS
LIN {X 0.159,Y -691.084,Z 362.485,A 0.000,B 0.000,C 90.000,E1 303.214} C_DIS
LIN {X -0.104,Y -692.641,Z 362.478,A 0.000,B 0.000,C 90.000,E1 302.054} C_DIS
LIN {X -0.353,Y -693.653,Z 362.473,A 0.000,B 0.000,C 90.000,E1 301.131} C_DIS
LIN {X 0.125,Y -694.044,Z 362.469,A 0.000,B 0.000,C 90.000,E1 300.384} C_DIS
LIN {X 0.142,Y -693.969,Z 362.462,A 0.000,B 0.000,C 90.000,E1 299.205} C_DIS
LIN {X -0.218,Y -693.910,Z 362.461,A 0.000,B 0.000,C 90.000,E1 298.999} C_DIS
LIN {X -0.088,Y -693.308,Z 362.457,A 0.000,B 0.000,C 90.000,E1 298.281} C_DIS
LIN {X 0.206,Y -691.723,Z 362.451,A 0.000,B 0.000,C 90.000,E1 297.078} C_DIS
LIN {X -0.131,Y -689.840,Z 362.444,A 0.000,B 0.000,C 90.000,E1 295.924} C_DIS
LIN {X 0.182,Y -687.984,Z 362.439,A 0.000,B 0.000,C 90.000,E1 294.951} C_DIS
LIN {X 0.111,Y -685.407,Z 362.432,A 0.000,B 0.000,C 90.000,E1 293.770} C_DIS
LIN {X 0.007,Y -682.663,Z 362.426,A 0.000,B 0.000,C 90.000,E1 292.589} C_DIS
LIN {X -0.142,Y -679.716,Z 362.419,A 0.000,B 0.000,C 90.000,E1 291.408} C_DIS
LIN {X 0.284,Y -676.760,Z 362.412,A 0.000,B 0.000,C 90.000,E1 290.174} C_DIS
LIN {X -0.281,Y -673.255,Z 362.404,A 0.000,B 0.000,C 90.000,E1 288.779} C_DIS
LIN {X 0.264,Y -667.457,Z 362.391,A 0.000,B 0.000,C 90.000,E1 286.315} C_DIS
LIN {X 0.337,Y -662.728,Z 362.379,A 0.000,B 0.000,C 90.000,E1 284.120} C_DIS
LIN {X 0.074,Y -656.591,Z 362.360,A 0.000,B 0.000,C 90.000,E1 280.715} C_DIS
LIN {X 0.231,Y -653.031,Z 362.345,A 0.000,B 0.000,C 90.000,E1 277.992} C_DIS
LIN {X -0.082,Y -651.016,Z 362.332,A 0.000,B 0.000,C 90.000,E1 275.796} C_DIS
LIN {X -0.150,Y -649.634,Z 362.318,A 0.000,B 0.000,C 90.000,E1 273.326} C_DIS
LIN {X -0.079,Y -648.994,Z 362.306,A 0.000,B 0.000,C 90.000,E1 271.088} C_DIS
LIN {X 0.185,Y -649.310,Z 362.287,A 0.000,B 0.000,C 90.000,E1 267.593} C_DIS
LIN {X 0.049,Y -650.016,Z 362.277,A 0.000,B 0.000,C 90.000,E1 265.869} C_DIS
LIN {X -0.123,Y -650.440,Z 362.272,A 0.000,B 0.000,C 90.000,E1 264.894} C_DIS
LIN {X 0.191,Y -650.999,Z 362.265,A 0.000,B 0.000,C 90.000,E1 263.628} C_DIS
LIN {X 0.217,Y -651.832,Z 362.255,A 0.000,B 0.000,C 90.000,E1 261.894} C_DIS
LIN {X -0.290,Y -652.214,Z 362.251,A 0.000,B 0.000,C 90.000,E1 261.197} C_DIS
LIN {X -0.149,Y -652.335,Z 362.247,A 0.000,B 0.000,C 90.000,E1 260.443} C_DIS
LIN {X -0.265,Y -652.354,Z 362.240,A 0.000,B 0.000,C 90.000,E1 259.218} C_DIS
LIN {X 0.005,Y -652.238,Z 362.230,A 0.000,B 0.000,C 90.000,E1 257.465} C_DIS
LIN {X 0.270,Y -651.989,Z 362.226,A 0.000,B 0.000,C 90.000,E1 256.700} C_DIS
LIN {X -0.225,Y -651.498,Z 362.221,A 0.000,B 0.000,C 90.000,E1 255.755} C_DIS
LIN {X 0.280,Y -651.233,Z 362.219,A 0.000,B 0.000,C 90.000,E1 255.463} C_DIS
LIN {X 0.027,Y -650.952,Z 362.217,A 0.000,B 0.000,C 90.000,E1 254.991} C_DIS
LIN {X -0.100,Y -650.748,Z 362.215,A 0.000,B 0.000,C 90.000,E1 254.755} C_DIS
LIN {X 0.181,Y -649.395,Z 362.210,A 0.000,B 0.000,C 90.000,E1 253.740} C_DIS
LIN {X -0.037,Y -648.148,Z 362.206,A 0.000,B 0.000,C 90.000,E1 253.015} C_DIS
LIN {X 0.356,Y -646.642,Z 362.202,A 0.000,B 0.000,C 90.000,E1 252.236} C_DIS
LIN {X 0.117,Y -644.883,Z 362.197,A 0.000,B 0.000,C 90.000,E1 251.511} C_DIS
LIN {X -0.139,Y -642.804,Z 362.193,A 0.000,B 0.000,C 90.000,E1 250.786} C_DIS
LIN {X 0.233,Y -639.584,Z 362.188,A 0.000,B 0.000,C 90.000,E1 249.752} C_DIS
LIN {X -0.040,Y -636.025,Z 362.182,A 0.000,B 0.000,C 90.000,E1 248.773} C_DIS
LIN {X -0.158,Y -633.320,Z 362.178,A 0.000,B 0.000,C 90.000,E1 248.028} C_DIS
LIN {X 0.064,Y -629.447,Z 362.172,A 0.000,B 0.000,C 90.000,E1 246.997} C_DIS
LIN {X -0.098,Y -624.408,Z 362.165,A 0.000,B 0.000,C 90.000,E1 245.741} C_DIS
LIN {X -0.080,Y -618.153,Z 362.157,A 0.000,B 0.000,C 90.000,E1 244.204} C_DIS
LIN {X -0.150,Y -612.851,Z 362.150,A 0.000,B 0.000,C 90.000,E1 242.922} C_DIS
LIN {X -0.314,Y -607.625,Z 362.142,A 0.000,B 0.000,C 90.000,E1 241.641} C_DIS
LIN {X -0.118,Y -600.253,Z 362.132,A 0.000,B 0.000,C 90.000,E1 239.793} C_DIS
LIN {X 0.206,Y -593.087,Z 362.122,A 0.000,B 0.000,C 90.000,E1 237.916} C_DIS
LIN {X 0.040,Y -585.340,Z 362.110,A 0.000,B 0.000,C 90.000,E1 235.801} C_DIS
LIN {X 0.319,Y -578.113,Z 362.098,A 0.000,B 0.000,C 90.000,E1 233.623} C_DIS
LIN {X 0.148,Y -574.481,Z 362.092,A 0.000,B 0.000,C 90.000,E1 232.557} C_DIS
LIN {X 0.095,Y -568.640,Z 362.083,A 0.000,B 0.000,C 90.000,E1 230.928} C_DIS
LIN {X -0.300,Y -561.078,Z 362.071,A 0.000,B 0.000,C 90.000,E1 228.771} C_DIS
LIN {X -0.342,Y -556.542,Z 362.063,A 0.000,B 0.000,C 90.000,E1 227.391} C_DIS
LIN {X -0.090,Y -552.012,Z 362.055,A 0.000,B 0.000,C 90.000,E1 225.972} C_DIS
LIN {X -0.314,Y -547.478,Z 362.048,A 0.000,B 0.000,C 90.000,E1 224.595} C_DIS
LIN {X 0.166,Y -542.101,Z 362.038,A 0.000,B 0.000,C 90.000,E1 222.852} C_DIS
LIN {X 0.155,Y -536.803,Z 362.029,A 0.000,B 0.000,C 90.000,E1 221.148} C_DIS
LIN {X 0.077,Y -530.767,Z 362.018,A 0.000,B 0.000,C 90.000,E1 219.152} C_DIS
LIN {X -0.121,Y -525.713,Z 362.008,A 0.000,B 0.000,C 90.000,E1 217.443} C_DIS
LIN {X -0.013,Y -519.312,Z 361.995,A 0.000,B 0.000,C 90.000,E1 215.105} C_DIS
LIN {X -0.044,Y -512.546,Z 361.980,A 0.000,B 0.000,C 90.000,E1 212.467} C_DIS
LIN {X 0.164,Y -508.391,Z 361.971,A 0.000,B 0.000,C 90.000,E1 210.669} C_DIS
LIN {X -0.097,Y -503.679,Z 361.959,A 0.000,B 0.000,C 90.000,E1 208.615} C_DIS
LIN {X -0.186,Y -500.376,Z 361.951,A 0.000,B 0.000,C 90.000,E1 207.129} C_DIS
LIN {X 0.109,Y -497.059,Z 361.942,A 0.000,B 0.000,C 90.000,E1 205.591} C_DIS
LIN {X 0.124,Y -493.694,Z 361.934,A 0.000,B 0.000,C 90.000,E1 204.079} C_DIS
LIN {X -0.083,Y -489.514,Z 361.924,A 0.000,B 0.000,C 90.000,E1 202.280} C_DIS
LIN {X 0.052,Y -485.903,Z 361.915,A 0.000,B 0.000,C 90.000,E1 200.737} C_DIS
LIN {X -0.053,Y -480.990,Z 361.903,A 0.000,B 0.000,C 90.000,E1 198.598} C_DIS
LIN {X -0.137,Y -476.318,Z 361.891,A 0.000,B 0.000,C 90.000,E1 196.441} C_DIS
LIN {X 0.160,Y -472.521,Z 361.881,A 0.000,B 0.000,C 90.000,E1 194.537} C_DIS
LIN {X 0.060,Y -468.300,Z 361.869,A 0.000,B 0.000,C 90.000,E1 192.355} C_DIS
LIN {X -0.149,Y -464.826,Z 361.858,A 0.000,B 0.000,C 90.000,E1 190.489} C_DIS
LIN {X -0.189,Y -460.981,Z 361.846,A 0.000,B 0.000,C 90.000,E1 188.276} C_DIS
LIN {X -0.069,Y -457.468,Z 361.833,A 0.000,B 0.000,C 90.000,E1 186.030} C_DIS
LIN {X -0.040,Y -454.303,Z 361.821,A 0.000,B 0.000,C 90.000,E1 183.784} C_DIS
LIN {X 0.037,Y -450.323,Z 361.801,A 0.000,B 0.000,C 90.000,E1 180.229} C_DIS
LIN {X -0.018,Y -447.123,Z 361.776,A 0.000,B 0.000,C 90.000,E1 175.698} C_DIS
LIN {X 0.089,Y -446.052,Z 361.754,A 0.000,B 0.000,C 90.000,E1 171.781} C_DIS
LIN {X 0.200,Y -446.247,Z 361.740,A 0.000,B 0.000,C 90.000,E1 169.162} C_DIS
LIN {X 0.050,Y -448.308,Z 361.715,A 0.000,B 0.000,C 90.000,E1 164.629} C_DIS
LIN {X 0.033,Y -450.166,Z 361.702,A 0.000,B 0.000,C 90.000,E1 162.362} C_DIS
LIN {X 0.014,Y -453.778,Z 361.684,A 0.000,B 0.000,C 90.000,E1 159.135} C_DIS
LIN {X 0.054,Y -457.405,Z 361.670,A 0.000,B 0.000,C 90.000,E1 156.561} C_DIS
LIN {X 0.071,Y -463.558,Z 361.650,A 0.000,B 0.000,C 90.000,E1 153.050} C_DIS
LIN {X 0.091,Y -472.796,Z 361.628,A 0.000,B 0.000,C 90.000,E1 148.948} C_DIS
LIN {X -0.009,Y -483.432,Z 361.607,A 0.000,B 0.000,C 90.000,E1 145.229} C_DIS
LIN {X 0.249,Y -490.411,Z 361.595,A 0.000,B 0.000,C 90.000,E1 143.050} C_DIS
LIN {X 0.176,Y -495.584,Z 361.586,A 0.000,B 0.000,C 90.000,E1 141.537} C_DIS
LIN {X -0.065,Y -499.615,Z 361.580,A 0.000,B 0.000,C 90.000,E1 140.356} C_DIS
LIN {X -0.045,Y -504.444,Z 361.571,A 0.000,B 0.000,C 90.000,E1 138.852} C_DIS
LIN {X 0.167,Y -508.147,Z 361.565,A 0.000,B 0.000,C 90.000,E1 137.634} C_DIS
LIN {X 0.057,Y -511.503,Z 361.558,A 0.000,B 0.000,C 90.000,E1 136.458} C_DIS
LIN {X 0.092,Y -513.782,Z 361.553,A 0.000,B 0.000,C 90.000,E1 135.567} C_DIS
LIN {X 0.155,Y -515.891,Z 361.548,A 0.000,B 0.000,C 90.000,E1 134.676} C_DIS
LIN {X 0.241,Y -517.693,Z 361.543,A 0.000,B 0.000,C 90.000,E1 133.785} C_DIS
LIN {X -0.013,Y -519.114,Z 361.539,A 0.000,B 0.000,C 90.000,E1 132.933} C_DIS
LIN {X 0.101,Y -520.280,Z 361.534,A 0.000,B 0.000,C 90.000,E1 132.043} C_DIS
LIN {X 0.263,Y -521.145,Z 361.529,A 0.000,B 0.000,C 90.000,E1 131.148} C_DIS
LIN {X -0.009,Y -521.648,Z 361.522,A 0.000,B 0.000,C 90.000,E1 130.011} C_DIS
LIN {X -0.109,Y -521.643,Z 361.519,A 0.000,B 0.000,C 90.000,E1 129.439} C_DIS
LIN {X 0.076,Y -521.332,Z 361.514,A 0.000,B 0.000,C 90.000,E1 128.543} C_DIS
LIN {X -0.067,Y -520.634,Z 361.509,A 0.000,B 0.000,C 90.000,E1 127.684} C_DIS
LIN {X -0.011,Y -518.934,Z 361.501,A 0.000,B 0.000,C 90.000,E1 126.217} C_DIS
LIN {X 0.178,Y -517.374,Z 361.495,A 0.000,B 0.000,C 90.000,E1 125.025} C_DIS
LIN {X 0.050,Y -516.463,Z 361.491,A 0.000,B 0.000,C 90.000,E1 124.452} C_DIS
LIN {X -0.091,Y -514.289,Z 361.485,A 0.000,B 0.000,C 90.000,E1 123.293} C_DIS
LIN {X -0.175,Y -512.532,Z 361.480,A 0.000,B 0.000,C 90.000,E1 122.418} C_DIS
LIN {X 0.067,Y -509.847,Z 361.473,A 0.000,B 0.000,C 90.000,E1 121.209} C_DIS
LIN {X 0.265,Y -506.932,Z 361.467,A 0.000,B 0.000,C 90.000,E1 120.001} C_DIS
LIN {X -0.151,Y -504.563,Z 361.462,A 0.000,B 0.000,C 90.000,E1 119.155} C_DIS
LIN {X 0.096,Y -502.056,Z 361.457,A 0.000,B 0.000,C 90.000,E1 118.231} C_DIS
LIN {X -0.028,Y -497.481,Z 361.449,A 0.000,B 0.000,C 90.000,E1 116.744} C_DIS
LIN {X -0.052,Y -493.541,Z 361.442,A 0.000,B 0.000,C 90.000,E1 115.540} C_DIS
LIN {X -0.167,Y -490.315,Z 361.437,A 0.000,B 0.000,C 90.000,E1 114.643} C_DIS
LIN {X 0.142,Y -485.695,Z 361.430,A 0.000,B 0.000,C 90.000,E1 113.387} C_DIS
LIN {X 0.185,Y -479.553,Z 361.422,A 0.000,B 0.000,C 90.000,E1 111.844} C_DIS
LIN {X 0.148,Y -472.819,Z 361.413,A 0.000,B 0.000,C 90.000,E1 110.301} C_DIS
LIN {X 0.211,Y -465.760,Z 361.404,A 0.000,B 0.000,C 90.000,E1 108.725} C_DIS
LIN {X -0.097,Y -461.217,Z 361.399,A 0.000,B 0.000,C 90.000,E1 107.764} C_DIS
LIN {X -0.137,Y -461.210,Z 361.399,A 0.000,B 0.000,C 90.000,E1 107.764} C_DIS
LIN {X -0.044,Y -467.655,Z 361.383,A 0.000,B 0.000,C 90.000,E1 104.954} C_DIS
LIN {X -0.031,Y -470.582,Z 361.373,A 0.000,B 0.000,C 90.000,E1 103.063} C_DIS
LIN {X -0.086,Y -475.873,Z 361.357,A 0.000,B 0.000,C 90.000,E1 100.254} C_DIS
LIN {X 0.221,Y -476.336,Z 361.355,A 0.000,B 0.000,C 90.000,E1 99.905} C_DIS
LIN {X 0.178,Y -481.843,Z 361.331,A 0.000,B 0.000,C 90.000,E1 95.568} C_DIS
LIN {X 0.025,Y -482.184,Z 361.329,A 0.000,B 0.000,C 90.000,E1 95.277} C_DIS
LIN {X -0.041,Y -485.343,Z 361.305,A 0.000,B 0.000,C 90.000,E1 90.974} C_DIS
LIN {X -0.217,Y -485.533,Z 361.304,A 0.000,B 0.000,C 90.000,E1 90.688} C_DIS
LIN {X -0.009,Y -486.336,Z 361.282,A 0.000,B 0.000,C 90.000,E1 86.674} C_DIS
LIN {X 0.125,Y -486.281,Z 361.278,A 0.000,B 0.000,C 90.000,E1 86.045} C_DIS
LIN {X -0.155,Y -484.694,Z 361.254,A 0.000,B 0.000,C 90.000,E1 81.781} C_DIS
LIN {X 0.193,Y -484.559,Z 361.253,A 0.000,B 0.000,C 90.000,E1 81.432} C_DIS
LIN {X 0.062,Y -480.498,Z 361.227,A 0.000,B 0.000,C 90.000,E1 76.825} C_DIS
LIN {X 0.199,Y -475.942,Z 361.210,A 0.000,B 0.000,C 90.000,E1 73.685} C_DIS
LIN {X 0.159,Y -475.958,Z 361.210,A 0.000,B 0.000,C 90.000,E1 73.685} C_DIS
LIN {X 0.204,Y -479.636,Z 361.206,A 0.000,B 0.000,C 90.000,E1 73.087} C_DIS
LIN {X -0.206,Y -484.202,Z 361.202,A 0.000,B 0.000,C 90.000,E1 72.362} C_DIS
LIN {X 0.062,Y -490.315,Z 361.196,A 0.000,B 0.000,C 90.000,E1 71.275} C_DIS
LIN {X -0.002,Y -495.259,Z 361.191,A 0.000,B 0.000,C 90.000,E1 70.369} C_DIS
LIN {X -0.105,Y -498.988,Z 361.187,A 0.000,B 0.000,C 90.000,E1 69.625} C_DIS
LIN {X 0.193,Y -503.668,Z 361.181,A 0.000,B 0.000,C 90.000,E1 68.539} C_DIS
LIN {X 0.231,Y -508.181,Z 361.174,A 0.000,B 0.000,C 90.000,E1 67.358} C_DIS
LIN {X 0.066,Y -511.493,Z 361.169,A 0.000,B 0.000,C 90.000,E1 66.485} C_DIS
LIN {X -0.182,Y -513.499,Z 361.166,A 0.000,B 0.000,C 90.000,E1 65.921} C_DIS
LIN {X 0.048,Y -517.239,Z 361.160,A 0.000,B 0.000,C 90.000,E1 64.717} C_DIS
LIN {X 0.009,Y -521.530,Z 361.151,A 0.000,B 0.000,C 90.000,E1 63.256} C_DIS
LIN {X -0.031,Y -526.440,Z 361.142,A 0.000,B 0.000,C 90.000,E1 61.513} C_DIS
LIN {X -0.018,Y -532.002,Z 361.131,A 0.000,B 0.000,C 90.000,E1 59.488} C_DIS
LIN {X -0.219,Y -535.932,Z 361.123,A 0.000,B 0.000,C 90.000,E1 58.074} C_DIS
LIN {X -0.057,Y -539.640,Z 361.115,A 0.000,B 0.000,C 90.000,E1 56.628} C_DIS
LIN {X 0.133,Y -541.797,Z 361.110,A 0.000,B 0.000,C 90.000,E1 55.754} C_DIS
LIN {X 0.236,Y -544.541,Z 361.104,A 0.000,B 0.000,C 90.000,E1 54.609} C_DIS
LIN {X 0.064,Y -546.978,Z 361.097,A 0.000,B 0.000,C 90.000,E1 53.497} C_DIS
LIN {X -0.189,Y -549.202,Z 361.091,A 0.000,B 0.000,C 90.000,E1 52.396} C_DIS
LIN {X -0.084,Y -550.167,Z 361.088,A 0.000,B 0.000,C 90.000,E1 51.823} C_DIS
LIN {X -0.231,Y -551.960,Z 361.080,A 0.000,B 0.000,C 90.000,E1 50.436} C_DIS
LIN {X -0.121,Y -552.645,Z 361.075,A 0.000,B 0.000,C 90.000,E1 49.585} C_DIS
LIN {X 0.057,Y -553.101,Z 361.071,A 0.000,B 0.000,C 90.000,E1 48.728} C_DIS
LIN {X -0.175,Y -553.199,Z 361.065,A 0.000,B 0.000,C 90.000,E1 47.634} C_DIS
LIN {X -0.047,Y -552.859,Z 361.060,A 0.000,B 0.000,C 90.000,E1 46.782} C_DIS
LIN {X -0.324,Y -552.310,Z 361.055,A 0.000,B 0.000,C 90.000,E1 45.972} C_DIS
LIN {X 0.176,Y -551.548,Z 361.051,A 0.000,B 0.000,C 90.000,E1 45.081} C_DIS
LIN {X -0.049,Y -549.976,Z 361.043,A 0.000,B 0.000,C 90.000,E1 43.704} C_DIS
LIN {X 0.089,Y -548.122,Z 361.035,A 0.000,B 0.000,C 90.000,E1 42.285} C_DIS
LIN {X -0.140,Y -545.893,Z 361.026,A 0.000,B 0.000,C 90.000,E1 40.620} C_DIS
LIN {X -0.062,Y -544.352,Z 361.019,A 0.000,B 0.000,C 90.000,E1 39.483} C_DIS
LIN {X -0.294,Y -542.094,Z 361.010,A 0.000,B 0.000,C 90.000,E1 37.810} C_DIS
LIN {X -0.141,Y -539.857,Z 361.000,A 0.000,B 0.000,C 90.000,E1 36.091} C_DIS
LIN {X 0.090,Y -537.629,Z 360.991,A 0.000,B 0.000,C 90.000,E1 34.358} C_DIS
LIN {X -0.175,Y -535.839,Z 360.983,A 0.000,B 0.000,C 90.000,E1 32.959} C_DIS
LIN {X -0.039,Y -534.077,Z 360.975,A 0.000,B 0.000,C 90.000,E1 31.514} C_DIS
LIN {X -0.060,Y -532.089,Z 360.966,A 0.000,B 0.000,C 90.000,E1 29.795} C_DIS
LIN {X 0.045,Y -529.863,Z 360.954,A 0.000,B 0.000,C 90.000,E1 27.769} C_DIS
LIN {X -0.087,Y -527.981,Z 360.945,A 0.000,B 0.000,C 90.000,E1 26.052} C_DIS
LIN {X -0.080,Y -526.039,Z 360.933,A 0.000,B 0.000,C 90.000,E1 24.027} C_DIS
LIN {X -0.179,Y -523.919,Z 360.921,A 0.000,B 0.000,C 90.000,E1 21.716} C_DIS
LIN {X 0.115,Y -522.617,Z 360.911,A 0.000,B 0.000,C 90.000,E1 19.939} C_DIS
LIN {X -0.144,Y -521.328,Z 360.900,A 0.000,B 0.000,C 90.000,E1 17.928} C_DIS
LIN {X -0.141,Y -520.161,Z 360.885,A 0.000,B 0.000,C 90.000,E1 15.300} C_DIS
LIN {X 0.061,Y -519.509,Z 360.869,A 0.000,B 0.000,C 90.000,E1 12.355} C_DIS
LIN {X -0.062,Y -519.616,Z 360.852,A 0.000,B 0.000,C 90.000,E1 9.443} C_DIS
LIN {X 0.260,Y -520.312,Z 360.838,A 0.000,B 0.000,C 90.000,E1 6.777} C_DIS
LIN {X -0.091,Y -521.746,Z 360.823,A 0.000,B 0.000,C 90.000,E1 4.188} C_DIS
LIN {X 0.004,Y -524.450,Z 360.805,A 0.000,B 0.000,C 90.000,E1 0.974} C_DIS
LIN {X 0.030,Y -527.985,Z 360.789,A 0.000,B 0.000,C 90.000,E1 358.051} C_DIS
LIN {X -0.112,Y -531.059,Z 360.778,A 0.000,B 0.000,C 90.000,E1 356.045} C_DIS
LIN {X -0.117,Y -534.528,Z 360.767,A 0.000,B 0.000,C 90.000,E1 354.033} C_DIS
LIN {X 0.207,Y -540.061,Z 360.751,A 0.000,B 0.000,C 90.000,E1 351.141} C_DIS
LIN {X -0.232,Y -545.966,Z 360.737,A 0.000,B 0.000,C 90.000,E1 348.634} C_DIS
LIN {X 0.161,Y -552.775,Z 360.723,A 0.000,B 0.000,C 90.000,E1 346.061} C_DIS
LIN {X 0.094,Y -557.660,Z 360.713,A 0.000,B 0.000,C 90.000,E1 344.393} C_DIS
LIN {X 0.138,Y -562.773,Z 360.704,A 0.000,B 0.000,C 90.000,E1 342.725} C_DIS
LIN {X 0.253,Y -568.746,Z 360.693,A 0.000,B 0.000,C 90.000,E1 340.786} C_DIS
LIN {X 0.153,Y -573.938,Z 360.684,A 0.000,B 0.000,C 90.000,E1 339.156} C_DIS
LIN {X 0.042,Y -580.807,Z 360.672,A 0.000,B 0.000,C 90.000,E1 336.997} C_DIS
LIN {X 0.298,Y -586.009,Z 360.663,A 0.000,B 0.000,C 90.000,E1 335.357} C_DIS
LIN {X 0.249,Y -590.416,Z 360.656,A 0.000,B 0.000,C 90.000,E1 334.024} C_DIS
LIN {X -0.259,Y -594.922,Z 360.648,A 0.000,B 0.000,C 90.000,E1 332.743} C_DIS
LIN {X 0.110,Y -599.450,Z 360.641,A 0.000,B 0.000,C 90.000,E1 331.385} C_DIS
LIN {X 0.136,Y -606.756,Z 360.629,A 0.000,B 0.000,C 90.000,E1 329.282} C_DIS
LIN {X 0.016,Y -610.379,Z 360.624,A 0.000,B 0.000,C 90.000,E1 328.250} C_DIS
LIN {X 0.168,Y -616.789,Z 360.614,A 0.000,B 0.000,C 90.000,E1 326.421} C_DIS
LIN {X -0.029,Y -622.328,Z 360.605,A 0.000,B 0.000,C 90.000,E1 324.895} C_DIS
LIN {X 0.065,Y -626.048,Z 360.599,A 0.000,B 0.000,C 90.000,E1 323.863} C_DIS
LIN {X 0.071,Y -629.707,Z 360.594,A 0.000,B 0.000,C 90.000,E1 322.844} C_DIS
LIN {X -0.387,Y -634.206,Z 360.587,A 0.000,B 0.000,C 90.000,E1 321.618} C_DIS
LIN {X 0.210,Y -642.443,Z 360.574,A 0.000,B 0.000,C 90.000,E1 319.299} C_DIS
LIN {X 0.022,Y -645.079,Z 360.570,A 0.000,B 0.000,C 90.000,E1 318.566} C_DIS
LIN {X 0.216,Y -648.448,Z 360.564,A 0.000,B 0.000,C 90.000,E1 317.553} C_DIS
LIN {X 0.277,Y -655.454,Z 360.553,A 0.000,B 0.000,C 90.000,E1 315.567} C_DIS
LIN {X 0.092,Y -660.569,Z 360.545,A 0.000,B 0.000,C 90.000,E1 314.109} C_DIS
LIN {X 0.005,Y -664.783,Z 360.538,A 0.000,B 0.000,C 90.000,E1 312.894} C_DIS
LIN {X 0.018,Y -668.209,Z 360.533,A 0.000,B 0.000,C 90.000,E1 311.919} C_DIS
LIN {X 0.096,Y -672.096,Z 360.526,A 0.000,B 0.000,C 90.000,E1 310.701} C_DIS
LIN {X 0.232,Y -675.964,Z 360.520,A 0.000,B 0.000,C 90.000,E1 309.483} C_DIS
LIN {X -0.408,Y -680.392,Z 360.512,A 0.000,B 0.000,C 90.000,E1 308.096} C_DIS
LIN {X -0.221,Y -682.406,Z 360.508,A 0.000,B 0.000,C 90.000,E1 307.363} C_DIS
LIN {X 0.151,Y -684.892,Z 360.502,A 0.000,B 0.000,C 90.000,E1 306.377} C_DIS
LIN {X 0.002,Y -687.219,Z 360.497,A 0.000,B 0.000,C 90.000,E1 305.438} C_DIS
LIN {X 0.046,Y -689.253,Z 360.492,A 0.000,B 0.000,C 90.000,E1 304.485} C_DIS
LIN {X -0.088,Y -690.624,Z 360.488,A 0.000,B 0.000,C 90.000,E1 303.785} C_DIS
LIN {X -0.212,Y -691.728,Z 360.484,A 0.000,B 0.000,C 90.000,E1 303.086} C_DIS
LIN {X -0.106,Y -692.938,Z 360.479,A 0.000,B 0.000,C 90.000,E1 302.133} C_DIS
LIN {X 0.006,Y -693.633,Z 360.475,A 0.000,B 0.000,C 90.000,E1 301.416} C_DIS
LIN {X -0.105,Y -693.968,Z 360.471,A 0.000,B 0.000,C 90.000,E1 300.718} C_DIS
LIN {X -0.221,Y -693.983,Z 360.468,A 0.000,B 0.000,C 90.000,E1 300.256} C_DIS
LIN {X 0.156,Y -693.760,Z 360.463,A 0.000,B 0.000,C 90.000,E1 299.283} C_DIS
LIN {X 0.044,Y -693.401,Z 360.460,A 0.000,B 0.000,C 90.000,E1 298.821} C_DIS
LIN {X -0.317,Y -693.066,Z 360.459,A 0.000,B 0.000,C 90.000,E1 298.615} C_DIS
LIN {X 0.174,Y -692.584,Z 360.456,A 0.000,B 0.000,C 90.000,E1 298.103} C_DIS
LIN {X -0.079,Y -691.237,Z 360.451,A 0.000,B 0.000,C 90.000,E1 297.180} C_DIS
LIN {X -0.052,Y -689.677,Z 360.446,A 0.000,B 0.000,C 90.000,E1 296.232} C_DIS
LIN {X -0.036,Y -687.817,Z 360.440,A 0.000,B 0.000,C 90.000,E1 295.283} C_DIS
LIN {X 0.177,Y -685.264,Z 360.434,A 0.000,B 0.000,C 90.000,E1 294.079} C_DIS
LIN {X 0.069,Y -682.497,Z 360.427,A 0.000,B 0.000,C 90.000,E1 292.898} C_DIS
LIN {X -0.083,Y -679.556,Z 360.421,A 0.000,B 0.000,C 90.000,E1 291.716} C_DIS
LIN {X -0.187,Y -675.349,Z 360.411,A 0.000,B 0.000,C 90.000,E1 290.047} C_DIS
LIN {X -0.142,Y -671.776,Z 360.403,A 0.000,B 0.000,C 90.000,E1 288.598} C_DIS
LIN {X 0.243,Y -666.571,Z 360.391,A 0.000,B 0.000,C 90.000,E1 286.386} C_DIS
LIN {X -0.333,Y -661.834,Z 360.379,A 0.000,B 0.000,C 90.000,E1 284.245} C_DIS
LIN {X -0.080,Y -655.287,Z 360.359,A 0.000,B 0.000,C 90.000,E1 280.546} C_DIS
LIN {X 0.309,Y -650.477,Z 360.335,A 0.000,B 0.000,C 90.000,E1 276.315} C_DIS
LIN {X 0.012,Y -649.094,Z 360.324,A 0.000,B 0.000,C 90.000,E1 274.359} C_DIS
LIN {X 0.287,Y -648.280,Z 360.313,A 0.000,B 0.000,C 90.000,E1 272.350} C_DIS
LIN {X 0.083,Y -647.901,Z 360.304,A 0.000,B 0.000,C 90.000,E1 270.630} C_DIS
LIN {X 0.086,Y -648.282,Z 360.287,A 0.000,B 0.000,C 90.000,E1 267.650} C_DIS
LIN {X -0.074,Y -649.004,Z 360.277,A 0.000,B 0.000,C 90.000,E1 265.927} C_DIS
LIN {X -0.222,Y -649.788,Z 360.268,A 0.000,B 0.000,C 90.000,E1 264.204} C_DIS
LIN {X 0.191,Y -650.748,Z 360.257,A 0.000,B 0.000,C 90.000,E1 262.186} C_DIS
LIN {X 0.175,Y -651.285,Z 360.251,A 0.000,B 0.000,C 90.000,E1 261.197} C_DIS
LIN {X -0.200,Y -651.483,Z 360.248,A 0.000,B 0.000,C 90.000,E1 260.735} C_DIS
LIN {X 0.177,Y -651.616,Z 360.240,A 0.000,B 0.000,C 90.000,E1 259.218} C_DIS
LIN {X 0.048,Y -651.770,Z 360.233,A 0.000,B 0.000,C 90.000,E1 257.993} C_DIS
LIN {X -0.203,Y -651.810,Z 360.231,A 0.000,B 0.000,C 90.000,E1 257.521} C_DIS
LIN {X 0.308,Y -651.722,Z 360.229,A 0.000,B 0.000,C 90.000,E1 257.229} C_DIS
LIN {X 0.184,Y -651.834,Z 360.228,A 0.000,B 0.000,C 90.000,E1 256.992} C_DIS
LIN {X 0.195,Y -651.557,Z 360.221,A 0.000,B 0.000,C 90.000,E1 255.755} C_DIS
LIN {X -0.181,Y -651.159,Z 360.217,A 0.000,B 0.000,C 90.000,E1 255.046} C_DIS
LIN {X 0.064,Y -650.459,Z 360.213,A 0.000,B 0.000,C 90.000,E1 254.283} C_DIS
LIN {X -0.018,Y -649.819,Z 360.210,A 0.000,B 0.000,C 90.000,E1 253.795} C_DIS
LIN {X 0.255,Y -648.209,Z 360.204,A 0.000,B 0.000,C 90.000,E1 252.779} C_DIS
LIN {X -0.116,Y -646.195,Z 360.199,A 0.000,B 0.000,C 90.000,E1 251.819} C_DIS
LIN {X -0.209,Y -645.079,Z 360.196,A 0.000,B 0.000,C 90.000,E1 251.329} C_DIS
LIN {X 0.144,Y -643.058,Z 360.192,A 0.000,B 0.000,C 90.000,E1 250.550} C_DIS
LIN {X -0.136,Y -640.766,Z 360.188,A 0.000,B 0.000,C 90.000,E1 249.826} C_DIS
LIN {X 0.279,Y -635.606,Z 360.180,A 0.000,B 0.000,C 90.000,E1 248.284} C_DIS
LIN {X 0.155,Y -632.854,Z 360.175,A 0.000,B 0.000,C 90.000,E1 247.539} C_DIS
LIN {X -0.194,Y -627.904,Z 360.168,A 0.000,B 0.000,C 90.000,E1 246.305} C_DIS
LIN {X -0.126,Y -623.873,Z 360.163,A 0.000,B 0.000,C 90.000,E1 245.281} C_DIS
LIN {X 0.185,Y -618.710,Z 360.156,A 0.000,B 0.000,C 90.000,E1 243.973} C_DIS
LIN {X 0.306,Y -610.355,Z 360.144,A 0.000,B 0.000,C 90.000,E1 241.897} C_DIS
LIN {X 0.380,Y -605.095,Z 360.137,A 0.000,B 0.000,C 90.000,E1 240.589} C_DIS
LIN {X -0.235,Y -598.912,Z 360.128,A 0.000,B 0.000,C 90.000,E1 239.076} C_DIS
LIN {X -0.156,Y -588.947,Z 360.113,A 0.000,B 0.000,C 90.000,E1 236.421} C_DIS
LIN {X 0.238,Y -579.797,Z 360.099,A 0.000,B 0.000,C 90.000,E1 233.703} C_DIS
LIN {X 0.087,Y -576.162,Z 360.093,A 0.000,B 0.000,C 90.000,E1 232.637} C_DIS
LIN {X -0.070,Y -571.299,Z 360.085,A 0.000,B 0.000,C 90.000,E1 231.295} C_DIS
LIN {X -0.285,Y -562.747,Z 360.071,A 0.000,B 0.000,C 90.000,E1 228.852} C_DIS
LIN {X 0.156,Y -557.294,Z 360.062,A 0.000,B 0.000,C 90.000,E1 227.148} C_DIS
LIN {X 0.033,Y -552.762,Z 360.054,A 0.000,B 0.000,C 90.000,E1 225.769} C_DIS
LIN {X 0.204,Y -548.224,Z 360.047,A 0.000,B 0.000,C 90.000,E1 224.352} C_DIS
LIN {X -0.095,Y -543.761,Z 360.039,A 0.000,B 0.000,C 90.000,E1 222.975} C_DIS
LIN {X -0.076,Y -538.452,Z 360.029,A 0.000,B 0.000,C 90.000,E1 221.272} C_DIS
LIN {X -0.121,Y -532.400,Z 360.018,A 0.000,B 0.000,C 90.000,E1 219.277} C_DIS
LIN {X 0.105,Y -526.486,Z 360.007,A 0.000,B 0.000,C 90.000,E1 217.237} C_DIS
LIN {X -0.141,Y -520.844,Z 359.996,A 0.000,B 0.000,C 90.000,E1 215.231} C_DIS
LIN {X -0.051,Y -514.782,Z 359.983,A 0.000,B 0.000,C 90.000,E1 212.880} C_DIS
LIN {X 0.010,Y -509.201,Z 359.970,A 0.000,B 0.000,C 90.000,E1 210.512} C_DIS
LIN {X -0.039,Y -504.518,Z 359.958,A 0.000,B 0.000,C 90.000,E1 208.437} C_DIS
LIN {X 0.186,Y -500.533,Z 359.948,A 0.000,B 0.000,C 90.000,E1 206.616} C_DIS
LIN {X -0.182,Y -497.252,Z 359.940,A 0.000,B 0.000,C 90.000,E1 205.155} C_DIS
LIN {X -0.208,Y -494.571,Z 359.933,A 0.000,B 0.000,C 90.000,E1 203.951} C_DIS
LIN {X 0.060,Y -490.420,Z 359.923,A 0.000,B 0.000,C 90.000,E1 202.099} C_DIS
LIN {X -0.267,Y -487.538,Z 359.916,A 0.000,B 0.000,C 90.000,E1 200.918} C_DIS
LIN {X 0.131,Y -482.650,Z 359.904,A 0.000,B 0.000,C 90.000,E1 198.725} C_DIS
LIN {X 0.094,Y -477.952,Z 359.892,A 0.000,B 0.000,C 90.000,E1 196.567} C_DIS
LIN {X -0.073,Y -473.533,Z 359.880,A 0.000,B 0.000,C 90.000,E1 194.411} C_DIS
LIN {X -0.058,Y -468.181,Z 359.864,A 0.000,B 0.000,C 90.000,E1 191.591} C_DIS
LIN {X 0.245,Y -463.601,Z 359.850,A 0.000,B 0.000,C 90.000,E1 189.029} C_DIS
LIN {X -0.214,Y -460.490,Z 359.840,A 0.000,B 0.000,C 90.000,E1 187.182} C_DIS
LIN {X 0.057,Y -455.787,Z 359.822,A 0.000,B 0.000,C 90.000,E1 183.955} C_DIS
LIN {X 0.191,Y -451.719,Z 359.802,A 0.000,B 0.000,C 90.000,E1 180.401} C_DIS
LIN {X 0.008,Y -449.109,Z 359.784,A 0.000,B 0.000,C 90.000,E1 177.192} C_DIS
LIN {X -0.026,Y -447.539,Z 359.765,A 0.000,B 0.000,C 90.000,E1 173.628} C_DIS
LIN {X 0.021,Y -447.346,Z 359.741,A 0.000,B 0.000,C 90.000,E1 169.398} C_DIS
LIN {X -0.076,Y -449.287,Z 359.716,A 0.000,B 0.000,C 90.000,E1 164.866} C_DIS
LIN {X 0.066,Y -452.676,Z 359.694,A 0.000,B 0.000,C 90.000,E1 160.967} C_DIS
LIN {X 0.219,Y -457.179,Z 359.675,A 0.000,B 0.000,C 90.000,E1 157.411} C_DIS
LIN {X -0.239,Y -463.541,Z 359.653,A 0.000,B 0.000,C 90.000,E1 153.640} C_DIS
LIN {X -0.233,Y -472.443,Z 359.631,A 0.000,B 0.000,C 90.000,E1 149.537} C_DIS
LIN {X -0.219,Y -482.816,Z 359.610,A 0.000,B 0.000,C 90.000,E1 145.801} C_DIS
LIN {X -0.148,Y -490.676,Z 359.596,A 0.000,B 0.000,C 90.000,E1 143.336} C_DIS
LIN {X -0.218,Y -495.792,Z 359.588,A 0.000,B 0.000,C 90.000,E1 141.823} C_DIS
LIN {X -0.072,Y -499.844,Z 359.581,A 0.000,B 0.000,C 90.000,E1 140.598} C_DIS
LIN {X -0.053,Y -504.653,Z 359.573,A 0.000,B 0.000,C 90.000,E1 139.094} C_DIS
LIN {X -0.217,Y -508.329,Z 359.566,A 0.000,B 0.000,C 90.000,E1 137.919} C_DIS
LIN {X 0.154,Y -510.902,Z 359.561,A 0.000,B 0.000,C 90.000,E1 136.986} C_DIS
LIN {X -0.170,Y -513.240,Z 359.556,A 0.000,B 0.000,C 90.000,E1 136.134} C_DIS
LIN {X -0.012,Y -514.692,Z 359.553,A 0.000,B 0.000,C 90.000,E1 135.526} C_DIS
LIN {X 0.055,Y -516.671,Z 359.548,A 0.000,B 0.000,C 90.000,E1 134.636} C_DIS
LIN {X -0.215,Y -518.363,Z 359.543,A 0.000,B 0.000,C 90.000,E1 133.785} C_DIS
LIN {X -0.011,Y -519.247,Z 359.540,A 0.000,B 0.000,C 90.000,E1 133.176} C_DIS
LIN {X 0.042,Y -520.670,Z 359.533,A 0.000,B 0.000,C 90.000,E1 132.000} C_DIS
LIN {X -0.121,Y -521.239,Z 359.530,A 0.000,B 0.000,C 90.000,E1 131.434} C_DIS
LIN {X 0.002,Y -521.820,Z 359.524,A 0.000,B 0.000,C 90.000,E1 130.253} C_DIS
LIN {X 0.189,Y -521.801,Z 359.519,A 0.000,B 0.000,C 90.000,E1 129.358} C_DIS
LIN {X -0.034,Y -521.382,Z 359.514,A 0.000,B 0.000,C 90.000,E1 128.508} C_DIS
LIN {X -0.182,Y -520.563,Z 359.509,A 0.000,B 0.000,C 90.000,E1 127.649} C_DIS
LIN {X -0.025,Y -518.738,Z 359.501,A 0.000,B 0.000,C 90.000,E1 126.171} C_DIS
LIN {X -0.257,Y -517.132,Z 359.494,A 0.000,B 0.000,C 90.000,E1 125.025} C_DIS
LIN {X 0.040,Y -516.225,Z 359.491,A 0.000,B 0.000,C 90.000,E1 124.405} C_DIS
LIN {X -0.098,Y -514.017,Z 359.485,A 0.000,B 0.000,C 90.000,E1 123.245} C_DIS
LIN {X 0.094,Y -512.281,Z 359.480,A 0.000,B 0.000,C 90.000,E1 122.339} C_DIS
LIN {X -0.109,Y -509.574,Z 359.473,A 0.000,B 0.000,C 90.000,E1 121.180} C_DIS
LIN {X 0.191,Y -507.529,Z 359.468,A 0.000,B 0.000,C 90.000,E1 120.256} C_DIS
LIN {X 0.095,Y -504.428,Z 359.462,A 0.000,B 0.000,C 90.000,E1 119.077} C_DIS
LIN {X -0.046,Y -501.136,Z 359.455,A 0.000,B 0.000,C 90.000,E1 117.897} C_DIS
LIN {X -0.077,Y -498.455,Z 359.450,A 0.000,B 0.000,C 90.000,E1 117.001} C_DIS
LIN {X -0.086,Y -494.619,Z 359.443,A 0.000,B 0.000,C 90.000,E1 115.796} C_DIS
LIN {X 0.217,Y -492.654,Z 359.440,A 0.000,B 0.000,C 90.000,E1 115.155} C_DIS
LIN {X 0.087,Y -489.382,Z 359.435,A 0.000,B 0.000,C 90.000,E1 114.259} C_DIS
LIN {X 0.186,Y -484.919,Z 359.428,A 0.000,B 0.000,C 90.000,E1 113.025} C_DIS
LIN {X 0.000,Y -479.525,Z 359.420,A 0.000,B 0.000,C 90.000,E1 111.663} C_DIS
LIN {X -0.223,Y -475.007,Z 359.414,A 0.000,B 0.000,C 90.000,E1 110.610} C_DIS
LIN {X 0.290,Y -468.873,Z 359.407,A 0.000,B 0.000,C 90.000,E1 109.141} C_DIS
LIN {X -0.052,Y -462.534,Z 359.399,A 0.000,B 0.000,C 90.000,E1 107.764} C_DIS
LIN {X -0.229,Y -461.636,Z 359.398,A 0.000,B 0.000,C 90.000,E1 107.583} C_DIS
LIN {X -0.268,Y -461.622,Z 359.398,A 0.000,B 0.000,C 90.000,E1 107.583} C_DIS
LIN {X 0.057,Y -467.757,Z 359.383,A 0.000,B 0.000,C 90.000,E1 104.898} C_DIS
LIN {X 0.029,Y -475.962,Z 359.357,A 0.000,B 0.000,C 90.000,E1 100.197} C_DIS
LIN {X 0.177,Y -476.676,Z 359.353,A 0.000,B 0.000,C 90.000,E1 99.557} C_DIS
LIN {X -0.176,Y -481.911,Z 359.331,A 0.000,B 0.000,C 90.000,E1 95.568} C_DIS
LIN {X 0.151,Y -482.202,Z 359.329,A 0.000,B 0.000,C 90.000,E1 95.220} C_DIS
LIN {X 0.089,Y -485.388,Z 359.305,A 0.000,B 0.000,C 90.000,E1 90.917} C_DIS
LIN {X -0.087,Y -485.529,Z 359.303,A 0.000,B 0.000,C 90.000,E1 90.630} C_DIS
LIN {X 0.122,Y -486.356,Z 359.281,A 0.000,B 0.000,C 90.000,E1 86.617} C_DIS
LIN {X -0.054,Y -486.368,Z 359.280,A 0.000,B 0.000,C 90.000,E1 86.331} C_DIS
LIN {X -0.064,Y -485.859,Z 359.275,A 0.000,B 0.000,C 90.000,E1 85.412} C_DIS
LIN {X -0.030,Y -484.693,Z 359.254,A 0.000,B 0.000,C 90.000,E1 81.724} C_DIS
LIN {X -0.162,Y -484.508,Z 359.252,A 0.000,B 0.000,C 90.000,E1 81.432} C_DIS
LIN {X 0.176,Y -480.441,Z 359.227,A 0.000,B 0.000,C 90.000,E1 76.769} C_DIS
LIN {X -0.164,Y -476.111,Z 359.210,A 0.000,B 0.000,C 90.000,E1 73.866} C_DIS
LIN {X -0.072,Y -476.111,Z 359.210,A 0.000,B 0.000,C 90.000,E1 73.850} C_DIS
LIN {X 0.236,Y -479.858,Z 359.207,A 0.000,B 0.000,C 90.000,E1 73.196} C_DIS
LIN {X 0.064,Y -483.454,Z 359.203,A 0.000,B 0.000,C 90.000,E1 72.598} C_DIS
LIN {X -0.074,Y -488.567,Z 359.198,A 0.000,B 0.000,C 90.000,E1 71.692} C_DIS
LIN {X -0.211,Y -490.135,Z 359.197,A 0.000,B 0.000,C 90.000,E1 71.402} C_DIS
LIN {X -0.156,Y -493.508,Z 359.193,A 0.000,B 0.000,C 90.000,E1 70.786} C_DIS
LIN {X -0.033,Y -497.951,Z 359.188,A 0.000,B 0.000,C 90.000,E1 69.880} C_DIS
LIN {X -0.040,Y -502.599,Z 359.182,A 0.000,B 0.000,C 90.000,E1 68.827} C_DIS
LIN {X -0.146,Y -503.895,Z 359.181,A 0.000,B 0.000,C 90.000,E1 68.539} C_DIS
LIN {X -0.269,Y -508.211,Z 359.174,A 0.000,B 0.000,C 90.000,E1 67.358} C_DIS
LIN {X 0.032,Y -511.274,Z 359.169,A 0.000,B 0.000,C 90.000,E1 66.433} C_DIS
LIN {X -0.010,Y -513.226,Z 359.166,A 0.000,B 0.000,C 90.000,E1 65.845} C_DIS
LIN {X 0.001,Y -516.856,Z 359.159,A 0.000,B 0.000,C 90.000,E1 64.665} C_DIS
LIN {X -0.142,Y -521.953,Z 359.150,A 0.000,B 0.000,C 90.000,E1 62.922} C_DIS
LIN {X -0.170,Y -526.846,Z 359.140,A 0.000,B 0.000,C 90.000,E1 61.179} C_DIS
LIN {X 0.155,Y -531.601,Z 359.130,A 0.000,B 0.000,C 90.000,E1 59.410} C_DIS
LIN {X -0.048,Y -535.536,Z 359.122,A 0.000,B 0.000,C 90.000,E1 57.995} C_DIS
LIN {X 0.112,Y -539.309,Z 359.114,A 0.000,B 0.000,C 90.000,E1 56.548} C_DIS
LIN {X 0.321,Y -542.152,Z 359.108,A 0.000,B 0.000,C 90.000,E1 55.388} C_DIS
LIN {X 0.087,Y -544.232,Z 359.103,A 0.000,B 0.000,C 90.000,E1 54.562} C_DIS
LIN {X 0.229,Y -546.717,Z 359.097,A 0.000,B 0.000,C 90.000,E1 53.417} C_DIS
LIN {X -0.024,Y -548.981,Z 359.091,A 0.000,B 0.000,C 90.000,E1 52.316} C_DIS
LIN {X 0.080,Y -550.011,Z 359.088,A 0.000,B 0.000,C 90.000,E1 51.743} C_DIS
LIN {X -0.067,Y -551.976,Z 359.080,A 0.000,B 0.000,C 90.000,E1 50.356} C_DIS
LIN {X -0.313,Y -552.736,Z 359.075,A 0.000,B 0.000,C 90.000,E1 49.542} C_DIS
LIN {X -0.192,Y -553.267,Z 359.070,A 0.000,B 0.000,C 90.000,E1 48.690} C_DIS
LIN {X -0.059,Y -553.447,Z 359.066,A 0.000,B 0.000,C 90.000,E1 47.838} C_DIS
LIN {X 0.051,Y -553.297,Z 359.063,A 0.000,B 0.000,C 90.000,E1 47.268} C_DIS
LIN {X 0.075,Y -553.353,Z 359.061,A 0.000,B 0.000,C 90.000,E1 46.986} C_DIS
LIN {X 0.205,Y -552.971,Z 359.056,A 0.000,B 0.000,C 90.000,E1 46.134} C_DIS
LIN {X 0.282,Y -552.490,Z 359.053,A 0.000,B 0.000,C 90.000,E1 45.567} C_DIS
LIN {X -0.070,Y -552.380,Z 359.052,A 0.000,B 0.000,C 90.000,E1 45.324} C_DIS
LIN {X 0.077,Y -551.329,Z 359.046,A 0.000,B 0.000,C 90.000,E1 44.190} C_DIS
LIN {X -0.215,Y -550.344,Z 359.041,A 0.000,B 0.000,C 90.000,E1 43.380} C_DIS
LIN {X -0.075,Y -548.951,Z 359.035,A 0.000,B 0.000,C 90.000,E1 42.243} C_DIS
LIN {X 0.080,Y -546.717,Z 359.025,A 0.000,B 0.000,C 90.000,E1 40.539} C_DIS
LIN {X 0.204,Y -544.791,Z 359.017,A 0.000,B 0.000,C 90.000,E1 39.116} C_DIS
LIN {X -0.020,Y -542.556,Z 359.008,A 0.000,B 0.000,C 90.000,E1 37.443} C_DIS
LIN {X 0.139,Y -540.327,Z 358.999,A 0.000,B 0.000,C 90.000,E1 35.724} C_DIS
LIN {X -0.072,Y -538.131,Z 358.989,A 0.000,B 0.000,C 90.000,E1 34.040} C_DIS
LIN {X -0.182,Y -536.324,Z 358.981,A 0.000,B 0.000,C 90.000,E1 32.625} C_DIS
LIN {X -0.037,Y -534.618,Z 358.973,A 0.000,B 0.000,C 90.000,E1 31.180} C_DIS
LIN {X -0.046,Y -532.629,Z 358.964,A 0.000,B 0.000,C 90.000,E1 29.461} C_DIS
LIN {X 0.118,Y -530.785,Z 358.954,A 0.000,B 0.000,C 90.000,E1 27.719} C_DIS
LIN {X 0.245,Y -528.916,Z 358.945,A 0.000,B 0.000,C 90.000,E1 25.976} C_DIS
LIN {X 0.264,Y -526.988,Z 358.933,A 0.000,B 0.000,C 90.000,E1 23.951} C_DIS
LIN {X 0.155,Y -524.647,Z 358.919,A 0.000,B 0.000,C 90.000,E1 21.354} C_DIS
LIN {X -0.024,Y -523.364,Z 358.909,A 0.000,B 0.000,C 90.000,E1 19.631} C_DIS
LIN {X 0.069,Y -522.175,Z 358.898,A 0.000,B 0.000,C 90.000,E1 17.583} C_DIS
LIN {X 0.119,Y -521.103,Z 358.883,A 0.000,B 0.000,C 90.000,E1 14.954} C_DIS
LIN {X -0.141,Y -520.594,Z 358.870,A 0.000,B 0.000,C 90.000,E1 12.647} C_DIS
LIN {X -0.138,Y -520.646,Z 358.854,A 0.000,B 0.000,C 90.000,E1 9.726} C_DIS
LIN {X 0.207,Y -521.198,Z 358.841,A 0.000,B 0.000,C 90.000,E1 7.352} C_DIS
LIN {X -0.001,Y -522.020,Z 358.831,A 0.000,B 0.000,C 90.000,E1 5.625} C_DIS
LIN {X 0.055,Y -524.760,Z 358.810,A 0.000,B 0.000,C 90.000,E1 1.835} C_DIS
LIN {X 0.064,Y -528.828,Z 358.791,A 0.000,B 0.000,C 90.000,E1 358.339} C_DIS
LIN {X 0.013,Y -529.962,Z 358.786,A 0.000,B 0.000,C 90.000,E1 357.478} C_DIS
LIN {X -0.056,Y -532.247,Z 358.778,A 0.000,B 0.000,C 90.000,E1 356.045} C_DIS
LIN {X -0.017,Y -535.252,Z 358.768,A 0.000,B 0.000,C 90.000,E1 354.318} C_DIS
LIN {X -0.266,Y -540.682,Z 358.753,A 0.000,B 0.000,C 90.000,E1 351.489} C_DIS
LIN {X 0.110,Y -544.418,Z 358.743,A 0.000,B 0.000,C 90.000,E1 349.746} C_DIS
LIN {X 0.145,Y -552.418,Z 358.726,A 0.000,B 0.000,C 90.000,E1 346.645} C_DIS
LIN {X -0.071,Y -557.250,Z 358.717,A 0.000,B 0.000,C 90.000,E1 344.991} C_DIS
LIN {X -0.129,Y -563.994,Z 358.704,A 0.000,B 0.000,C 90.000,E1 342.779} C_DIS
LIN {X 0.175,Y -570.866,Z 358.692,A 0.000,B 0.000,C 90.000,E1 340.550} C_DIS
LIN {X -0.051,Y -575.203,Z 358.685,A 0.000,B 0.000,C 90.000,E1 339.209} C_DIS
LIN {X -0.121,Y -582.091,Z 358.672,A 0.000,B 0.000,C 90.000,E1 337.050} C_DIS
LIN {X 0.051,Y -588.196,Z 358.662,A 0.000,B 0.000,C 90.000,E1 335.153} C_DIS
LIN {X 0.044,Y -592.629,Z 358.655,A 0.000,B 0.000,C 90.000,E1 333.819} C_DIS
LIN {X 0.196,Y -596.288,Z 358.649,A 0.000,B 0.000,C 90.000,E1 332.743} C_DIS
LIN {X 0.066,Y -600.806,Z 358.641,A 0.000,B 0.000,C 90.000,E1 331.435} C_DIS
LIN {X 0.139,Y -608.139,Z 358.630,A 0.000,B 0.000,C 90.000,E1 329.331} C_DIS
LIN {X -0.277,Y -611.768,Z 358.624,A 0.000,B 0.000,C 90.000,E1 328.329} C_DIS
LIN {X 0.205,Y -619.123,Z 358.612,A 0.000,B 0.000,C 90.000,E1 326.215} C_DIS
LIN {X -0.277,Y -623.744,Z 358.605,A 0.000,B 0.000,C 90.000,E1 324.975} C_DIS
LIN {X 0.202,Y -627.425,Z 358.600,A 0.000,B 0.000,C 90.000,E1 323.909} C_DIS
LIN {X 0.213,Y -631.869,Z 358.593,A 0.000,B 0.000,C 90.000,E1 322.637} C_DIS
LIN {X 0.185,Y -636.352,Z 358.586,A 0.000,B 0.000,C 90.000,E1 321.376} C_DIS
LIN {X -0.043,Y -644.454,Z 358.573,A 0.000,B 0.000,C 90.000,E1 319.138} C_DIS
LIN {X 0.132,Y -648.632,Z 358.566,A 0.000,B 0.000,C 90.000,E1 317.877} C_DIS
LIN {X 0.190,Y -655.502,Z 358.555,A 0.000,B 0.000,C 90.000,E1 315.891} C_DIS
LIN {X 0.057,Y -658.894,Z 358.550,A 0.000,B 0.000,C 90.000,E1 314.919} C_DIS
LIN {X -0.079,Y -664.736,Z 358.540,A 0.000,B 0.000,C 90.000,E1 313.218} C_DIS
LIN {X -0.066,Y -668.899,Z 358.533,A 0.000,B 0.000,C 90.000,E1 312.000} C_DIS
LIN {X 0.022,Y -672.715,Z 358.527,A 0.000,B 0.000,C 90.000,E1 310.782} C_DIS
LIN {X -0.243,Y -677.203,Z 358.519,A 0.000,B 0.000,C 90.000,E1 309.358} C_DIS
LIN {X -0.038,Y -680.802,Z 358.512,A 0.000,B 0.000,C 90.000,E1 308.141} C_DIS
LIN {X 0.304,Y -683.418,Z 358.507,A 0.000,B 0.000,C 90.000,E1 307.156} C_DIS
LIN {X 0.139,Y -685.797,Z 358.501,A 0.000,B 0.000,C 90.000,E1 306.217} C_DIS
LIN {X -0.401,Y -687.897,Z 358.496,A 0.000,B 0.000,C 90.000,E1 305.311} C_DIS
LIN {X 0.019,Y -689.341,Z 358.492,A 0.000,B 0.000,C 90.000,E1 304.565} C_DIS
LIN {X -0.112,Y -690.655,Z 358.488,A 0.000,B 0.000,C 90.000,E1 303.865} C_DIS
LIN {X 0.365,Y -692.035,Z 358.483,A 0.000,B 0.000,C 90.000,E1 302.880} C_DIS
LIN {X 0.108,Y -693.171,Z 358.478,A 0.000,B 0.000,C 90.000,E1 301.957} C_DIS
LIN {X -0.003,Y -693.775,Z 358.474,A 0.000,B 0.000,C 90.000,E1 301.258} C_DIS
LIN {X 0.122,Y -693.971,Z 358.470,A 0.000,B 0.000,C 90.000,E1 300.541} C_DIS
LIN {X -0.345,Y -693.757,Z 358.466,A 0.000,B 0.000,C 90.000,E1 299.873} C_DIS
LIN {X 0.149,Y -693.515,Z 358.463,A 0.000,B 0.000,C 90.000,E1 299.361} C_DIS
LIN {X 0.037,Y -693.108,Z 358.461,A 0.000,B 0.000,C 90.000,E1 298.899} C_DIS
LIN {X 0.044,Y -691.537,Z 358.454,A 0.000,B 0.000,C 90.000,E1 297.719} C_DIS
LIN {X -0.060,Y -689.069,Z 358.446,A 0.000,B 0.000,C 90.000,E1 296.309} C_DIS
LIN {X 0.019,Y -687.701,Z 358.442,A 0.000,B 0.000,C 90.000,E1 295.591} C_DIS
LIN {X 0.163,Y -684.540,Z 358.434,A 0.000,B 0.000,C 90.000,E1 294.155} C_DIS
LIN {X 0.316,Y -681.748,Z 358.428,A 0.000,B 0.000,C 90.000,E1 292.950} C_DIS
LIN {X 0.082,Y -678.159,Z 358.420,A 0.000,B 0.000,C 90.000,E1 291.535} C_DIS
LIN {X -0.216,Y -674.518,Z 358.412,A 0.000,B 0.000,C 90.000,E1 290.120} C_DIS
LIN {X -0.178,Y -670.876,Z 358.404,A 0.000,B 0.000,C 90.000,E1 288.671} C_DIS
LIN {X -0.252,Y -665.652,Z 358.392,A 0.000,B 0.000,C 90.000,E1 286.496} C_DIS
LIN {X 0.143,Y -662.922,Z 358.385,A 0.000,B 0.000,C 90.000,E1 285.245} C_DIS
LIN {X 0.030,Y -658.933,Z 358.374,A 0.000,B 0.000,C 90.000,E1 283.300} C_DIS
LIN {X -0.147,Y -653.954,Z 358.358,A 0.000,B 0.000,C 90.000,E1 280.366} C_DIS
LIN {X 0.302,Y -649.487,Z 358.336,A 0.000,B 0.000,C 90.000,E1 276.372} C_DIS
LIN {X -0.246,Y -647.961,Z 358.323,A 0.000,B 0.000,C 90.000,E1 274.188} C_DIS
LIN {X 0.003,Y -647.194,Z 358.312,A 0.000,B 0.000,C 90.000,E1 272.178} C_DIS
LIN {X -0.225,Y -646.848,Z 358.302,A 0.000,B 0.000,C 90.000,E1 270.458} C_DIS
LIN {X -0.041,Y -647.237,Z 358.287,A 0.000,B 0.000,C 90.000,E1 267.707} C_DIS
LIN {X -0.270,Y -647.978,Z 358.278,A 0.000,B 0.000,C 90.000,E1 265.988} C_DIS
LIN {X 0.090,Y -648.908,Z 358.267,A 0.000,B 0.000,C 90.000,E1 263.970} C_DIS
LIN {X -0.154,Y -649.888,Z 358.256,A 0.000,B 0.000,C 90.000,E1 262.008} C_DIS
LIN {X 0.227,Y -650.593,Z 358.249,A 0.000,B 0.000,C 90.000,E1 260.735} C_DIS
LIN {X -0.173,Y -650.892,Z 358.240,A 0.000,B 0.000,C 90.000,E1 259.285} C_DIS
LIN {X 0.320,Y -651.282,Z 358.232,A 0.000,B 0.000,C 90.000,E1 257.757} C_DIS
LIN {X -0.331,Y -651.589,Z 358.227,A 0.000,B 0.000,C 90.000,E1 256.825} C_DIS
LIN {X -0.078,Y -651.541,Z 358.223,A 0.000,B 0.000,C 90.000,E1 256.061} C_DIS
LIN {X 0.335,Y -651.296,Z 358.218,A 0.000,B 0.000,C 90.000,E1 255.283} C_DIS
LIN {X -0.045,Y -650.774,Z 358.214,A 0.000,B 0.000,C 90.000,E1 254.574} C_DIS
LIN {X -0.303,Y -650.281,Z 358.212,A 0.000,B 0.000,C 90.000,E1 254.102} C_DIS
LIN {X -0.029,Y -649.056,Z 358.206,A 0.000,B 0.000,C 90.000,E1 253.087} C_DIS
LIN {X 0.279,Y -646.867,Z 358.199,A 0.000,B 0.000,C 90.000,E1 251.819} C_DIS
LIN {X 0.039,Y -645.266,Z 358.195,A 0.000,B 0.000,C 90.000,E1 251.094} C_DIS
LIN {X -0.216,Y -643.311,Z 358.191,A 0.000,B 0.000,C 90.000,E1 250.369} C_DIS
LIN {X -0.324,Y -641.894,Z 358.188,A 0.000,B 0.000,C 90.000,E1 249.880} C_DIS
LIN {X 0.122,Y -636.939,Z 358.180,A 0.000,B 0.000,C 90.000,E1 248.337} C_DIS
LIN {X -0.226,Y -634.272,Z 358.176,A 0.000,B 0.000,C 90.000,E1 247.614} C_DIS
LIN {X -0.306,Y -629.362,Z 358.169,A 0.000,B 0.000,C 90.000,E1 246.357} C_DIS
LIN {X 0.095,Y -625.393,Z 358.163,A 0.000,B 0.000,C 90.000,E1 245.305} C_DIS
LIN {X 0.130,Y -619.224,Z 358.154,A 0.000,B 0.000,C 90.000,E1 243.768} C_DIS
LIN {X 0.019,Y -611.980,Z 358.144,A 0.000,B 0.000,C 90.000,E1 241.975} C_DIS
LIN {X 0.117,Y -606.774,Z 358.137,A 0.000,B 0.000,C 90.000,E1 240.667} C_DIS
LIN {X -0.234,Y -599.568,Z 358.127,A 0.000,B 0.000,C 90.000,E1 238.869} C_DIS
LIN {X -0.336,Y -590.617,Z 358.114,A 0.000,B 0.000,C 90.000,E1 236.501} C_DIS
LIN {X -0.178,Y -580.587,Z 358.097,A 0.000,B 0.000,C 90.000,E1 233.543} C_DIS
LIN {X 0.145,Y -576.848,Z 358.091,A 0.000,B 0.000,C 90.000,E1 232.431} C_DIS
LIN {X -0.148,Y -572.954,Z 358.085,A 0.000,B 0.000,C 90.000,E1 231.376} C_DIS
LIN {X 0.006,Y -565.294,Z 358.073,A 0.000,B 0.000,C 90.000,E1 229.175} C_DIS
LIN {X -0.297,Y -559.850,Z 358.064,A 0.000,B 0.000,C 90.000,E1 227.553} C_DIS
LIN {X -0.328,Y -554.418,Z 358.055,A 0.000,B 0.000,C 90.000,E1 225.891} C_DIS
LIN {X -0.089,Y -548.964,Z 358.046,A 0.000,B 0.000,C 90.000,E1 224.190} C_DIS
LIN {X -0.001,Y -545.408,Z 358.039,A 0.000,B 0.000,C 90.000,E1 223.056} C_DIS
LIN {X 0.052,Y -540.071,Z 358.030,A 0.000,B 0.000,C 90.000,E1 221.353} C_DIS
LIN {X 0.048,Y -534.018,Z 358.019,A 0.000,B 0.000,C 90.000,E1 219.358} C_DIS
LIN {X -0.102,Y -528.060,Z 358.008,A 0.000,B 0.000,C 90.000,E1 217.363} C_DIS
LIN {X 0.112,Y -522.371,Z 357.996,A 0.000,B 0.000,C 90.000,E1 215.311} C_DIS
LIN {X -0.118,Y -517.025,Z 357.985,A 0.000,B 0.000,C 90.000,E1 213.293} C_DIS
LIN {X 0.097,Y -510.670,Z 357.970,A 0.000,B 0.000,C 90.000,E1 210.620} C_DIS
LIN {X -0.095,Y -505.994,Z 357.959,A 0.000,B 0.000,C 90.000,E1 208.565} C_DIS
LIN {X 0.093,Y -502.661,Z 357.950,A 0.000,B 0.000,C 90.000,E1 207.052} C_DIS
LIN {X -0.242,Y -499.447,Z 357.942,A 0.000,B 0.000,C 90.000,E1 205.591} C_DIS
LIN {X -0.179,Y -496.134,Z 357.934,A 0.000,B 0.000,C 90.000,E1 204.079} C_DIS
LIN {X -0.144,Y -491.999,Z 357.924,A 0.000,B 0.000,C 90.000,E1 202.259} C_DIS
LIN {X -0.177,Y -489.158,Z 357.917,A 0.000,B 0.000,C 90.000,E1 201.046} C_DIS
LIN {X -0.190,Y -484.268,Z 357.905,A 0.000,B 0.000,C 90.000,E1 198.906} C_DIS
LIN {X -0.043,Y -479.545,Z 357.893,A 0.000,B 0.000,C 90.000,E1 196.732} C_DIS
LIN {X -0.138,Y -475.738,Z 357.883,A 0.000,B 0.000,C 90.000,E1 194.883} C_DIS
LIN {X 0.077,Y -472.668,Z 357.874,A 0.000,B 0.000,C 90.000,E1 193.300} C_DIS
LIN {X 0.063,Y -469.187,Z 357.864,A 0.000,B 0.000,C 90.000,E1 191.422} C_DIS
LIN {X 0.143,Y -465.140,Z 357.851,A 0.000,B 0.000,C 90.000,E1 189.208} C_DIS
LIN {X -0.215,Y -462.030,Z 357.841,A 0.000,B 0.000,C 90.000,E1 187.352} C_DIS
LIN {X -0.111,Y -457.699,Z 357.825,A 0.000,B 0.000,C 90.000,E1 184.473} C_DIS
LIN {X 0.126,Y -453.434,Z 357.805,A 0.000,B 0.000,C 90.000,E1 180.917} C_DIS
LIN {X 0.170,Y -450.453,Z 357.786,A 0.000,B 0.000,C 90.000,E1 177.364} C_DIS
LIN {X -0.112,Y -448.682,Z 357.764,A 0.000,B 0.000,C 90.000,E1 173.514} C_DIS
LIN {X -0.017,Y -448.527,Z 357.741,A 0.000,B 0.000,C 90.000,E1 169.285} C_DIS
LIN {X -0.065,Y -450.476,Z 357.715,A 0.000,B 0.000,C 90.000,E1 164.755} C_DIS
LIN {X 0.114,Y -453.887,Z 357.694,A 0.000,B 0.000,C 90.000,E1 160.859} C_DIS
LIN {X -0.123,Y -458.379,Z 357.674,A 0.000,B 0.000,C 90.000,E1 157.358} C_DIS
LIN {X 0.003,Y -465.339,Z 357.651,A 0.000,B 0.000,C 90.000,E1 153.204} C_DIS
LIN {X 0.149,Y -473.683,Z 357.630,A 0.000,B 0.000,C 90.000,E1 149.410} C_DIS
LIN {X 0.224,Y -484.093,Z 357.609,A 0.000,B 0.000,C 90.000,E1 145.674} C_DIS
LIN {X -0.061,Y -491.966,Z 357.596,A 0.000,B 0.000,C 90.000,E1 143.256} C_DIS
LIN {X -0.242,Y -498.056,Z 357.586,A 0.000,B 0.000,C 90.000,E1 141.457} C_DIS
LIN {X 0.064,Y -501.050,Z 357.581,A 0.000,B 0.000,C 90.000,E1 140.517} C_DIS
LIN {X 0.224,Y -504.913,Z 357.574,A 0.000,B 0.000,C 90.000,E1 139.299} C_DIS
LIN {X -0.269,Y -508.521,Z 357.567,A 0.000,B 0.000,C 90.000,E1 138.162} C_DIS
LIN {X 0.102,Y -511.171,Z 357.563,A 0.000,B 0.000,C 90.000,E1 137.229} C_DIS
LIN {X -0.221,Y -513.498,Z 357.558,A 0.000,B 0.000,C 90.000,E1 136.377} C_DIS
LIN {X -0.165,Y -515.582,Z 357.553,A 0.000,B 0.000,C 90.000,E1 135.486} C_DIS
LIN {X 0.009,Y -516.901,Z 357.549,A 0.000,B 0.000,C 90.000,E1 134.879} C_DIS
LIN {X -0.260,Y -518.567,Z 357.544,A 0.000,B 0.000,C 90.000,E1 134.028} C_DIS
LIN {X -0.149,Y -519.850,Z 357.540,A 0.000,B 0.000,C 90.000,E1 133.137} C_DIS
LIN {X 0.067,Y -520.353,Z 357.536,A 0.000,B 0.000,C 90.000,E1 132.528} C_DIS
LIN {X 0.290,Y -521.044,Z 357.533,A 0.000,B 0.000,C 90.000,E1 131.919} C_DIS
LIN {X -0.215,Y -521.459,Z 357.530,A 0.000,B 0.000,C 90.000,E1 131.391} C_DIS
LIN {X -0.031,Y -521.833,Z 357.525,A 0.000,B 0.000,C 90.000,E1 130.496} C_DIS
LIN {X 0.040,Y -521.702,Z 357.519,A 0.000,B 0.000,C 90.000,E1 129.322} C_DIS
LIN {X -0.107,Y -521.198,Z 357.514,A 0.000,B 0.000,C 90.000,E1 128.463} C_DIS
LIN {X 0.065,Y -520.314,Z 357.509,A 0.000,B 0.000,C 90.000,E1 127.569} C_DIS
LIN {X 0.157,Y -518.049,Z 357.499,A 0.000,B 0.000,C 90.000,E1 125.804} C_DIS
LIN {X -0.091,Y -516.385,Z 357.493,A 0.000,B 0.000,C 90.000,E1 124.659} C_DIS
LIN {X -0.233,Y -514.240,Z 357.486,A 0.000,B 0.000,C 90.000,E1 123.499} C_DIS
LIN {X 0.032,Y -511.931,Z 357.479,A 0.000,B 0.000,C 90.000,E1 122.291} C_DIS
LIN {X -0.171,Y -509.217,Z 357.473,A 0.000,B 0.000,C 90.000,E1 121.131} C_DIS
LIN {X 0.129,Y -507.191,Z 357.468,A 0.000,B 0.000,C 90.000,E1 120.207} C_DIS
LIN {X 0.034,Y -504.110,Z 357.461,A 0.000,B 0.000,C 90.000,E1 119.027} C_DIS
LIN {X -0.105,Y -500.843,Z 357.455,A 0.000,B 0.000,C 90.000,E1 117.847} C_DIS
LIN {X 0.090,Y -498.248,Z 357.450,A 0.000,B 0.000,C 90.000,E1 116.924} C_DIS
LIN {X 0.072,Y -494.595,Z 357.443,A 0.000,B 0.000,C 90.000,E1 115.720} C_DIS
LIN {X -0.035,Y -491.660,Z 357.438,A 0.000,B 0.000,C 90.000,E1 114.823} C_DIS
LIN {X 0.096,Y -487.449,Z 357.431,A 0.000,B 0.000,C 90.000,E1 113.590} C_DIS
LIN {X -0.079,Y -481.865,Z 357.423,A 0.000,B 0.000,C 90.000,E1 112.078} C_DIS
LIN {X 0.153,Y -476.433,Z 357.415,A 0.000,B 0.000,C 90.000,E1 110.663} C_DIS
LIN {X 0.087,Y -470.508,Z 357.407,A 0.000,B 0.000,C 90.000,E1 109.268} C_DIS
LIN {X 0.105,Y -463.561,Z 357.398,A 0.000,B 0.000,C 90.000,E1 107.692} C_DIS
LIN {X 0.095,Y -462.035,Z 357.396,A 0.000,B 0.000,C 90.000,E1 107.347} C_DIS
LIN {X 0.055,Y -462.038,Z 357.396,A 0.000,B 0.000,C 90.000,E1 107.347} C_DIS
LIN {X 0.213,Y -467.857,Z 357.383,A 0.000,B 0.000,C 90.000,E1 104.828} C_DIS
LIN {X -0.227,Y -475.415,Z 357.358,A 0.000,B 0.000,C 90.000,E1 100.489} C_DIS
LIN {X 0.079,Y -476.067,Z 357.356,A 0.000,B 0.000,C 90.000,E1 100.141} C_DIS
LIN {X -0.116,Y -481.992,Z 357.331,A 0.000,B 0.000,C 90.000,E1 95.511} C_DIS
LIN {X 0.018,Y -482.360,Z 357.327,A 0.000,B 0.000,C 90.000,E1 94.878} C_DIS
LIN {X 0.154,Y -485.441,Z 357.305,A 0.000,B 0.000,C 90.000,E1 90.859} C_DIS
LIN {X -0.194,Y -485.505,Z 357.302,A 0.000,B 0.000,C 90.000,E1 90.286} C_DIS
LIN {X 0.187,Y -486.379,Z 357.281,A 0.000,B 0.000,C 90.000,E1 86.560} C_DIS
LIN {X 0.012,Y -486.366,Z 357.279,A 0.000,B 0.000,C 90.000,E1 86.274} C_DIS
LIN {X 0.100,Y -484.690,Z 357.254,A 0.000,B 0.000,C 90.000,E1 81.659} C_DIS
LIN {X -0.233,Y -484.081,Z 357.250,A 0.000,B 0.000,C 90.000,E1 81.084} C_DIS
LIN {X -0.098,Y -480.644,Z 357.228,A 0.000,B 0.000,C 90.000,E1 77.061} C_DIS
LIN {X -0.132,Y -480.358,Z 357.226,A 0.000,B 0.000,C 90.000,E1 76.756} C_DIS
LIN {X 0.119,Y -476.291,Z 357.211,A 0.000,B 0.000,C 90.000,E1 73.976} C_DIS
LIN {X 0.079,Y -476.319,Z 357.211,A 0.000,B 0.000,C 90.000,E1 73.976} C_DIS
LIN {X -0.157,Y -479.263,Z 357.208,A 0.000,B 0.000,C 90.000,E1 73.504} C_DIS
LIN {X 0.118,Y -484.432,Z 357.203,A 0.000,B 0.000,C 90.000,E1 72.543} C_DIS
LIN {X 0.213,Y -488.581,Z 357.199,A 0.000,B 0.000,C 90.000,E1 71.764} C_DIS
LIN {X 0.182,Y -490.683,Z 357.196,A 0.000,B 0.000,C 90.000,E1 71.329} C_DIS
LIN {X 0.236,Y -493.605,Z 357.193,A 0.000,B 0.000,C 90.000,E1 70.786} C_DIS
LIN {X -0.120,Y -497.755,Z 357.189,A 0.000,B 0.000,C 90.000,E1 69.934} C_DIS
LIN {X -0.089,Y -500.823,Z 357.184,A 0.000,B 0.000,C 90.000,E1 69.209} C_DIS
LIN {X 0.051,Y -503.293,Z 357.181,A 0.000,B 0.000,C 90.000,E1 68.592} C_DIS
LIN {X -0.167,Y -506.583,Z 357.176,A 0.000,B 0.000,C 90.000,E1 67.720} C_DIS
LIN {X 0.020,Y -508.706,Z 357.173,A 0.000,B 0.000,C 90.000,E1 67.102} C_DIS
LIN {X -0.030,Y -512.520,Z 357.166,A 0.000,B 0.000,C 90.000,E1 65.921} C_DIS
LIN {X -0.156,Y -516.964,Z 357.158,A 0.000,B 0.000,C 90.000,E1 64.460} C_DIS
LIN {X 0.173,Y -522.018,Z 357.148,A 0.000,B 0.000,C 90.000,E1 62.666} C_DIS
LIN {X -0.254,Y -526.095,Z 357.140,A 0.000,B 0.000,C 90.000,E1 61.257} C_DIS
LIN {X 0.013,Y -531.648,Z 357.129,A 0.000,B 0.000,C 90.000,E1 59.203} C_DIS
LIN {X -0.187,Y -535.563,Z 357.121,A 0.000,B 0.000,C 90.000,E1 57.788} C_DIS
LIN {X -0.033,Y -538.648,Z 357.115,A 0.000,B 0.000,C 90.000,E1 56.628} C_DIS
LIN {X 0.183,Y -542.220,Z 357.107,A 0.000,B 0.000,C 90.000,E1 55.182} C_DIS
LIN {X -0.052,Y -544.263,Z 357.102,A 0.000,B 0.000,C 90.000,E1 54.356} C_DIS
LIN {X 0.129,Y -547.342,Z 357.094,A 0.000,B 0.000,C 90.000,E1 52.924} C_DIS
LIN {X -0.116,Y -549.598,Z 357.088,A 0.000,B 0.000,C 90.000,E1 51.823} C_DIS
LIN {X 0.099,Y -551.258,Z 357.082,A 0.000,B 0.000,C 90.000,E1 50.678} C_DIS
LIN {X 0.139,Y -551.995,Z 357.079,A 0.000,B 0.000,C 90.000,E1 50.114} C_DIS
LIN {X -0.046,Y -553.041,Z 357.072,A 0.000,B 0.000,C 90.000,E1 49.013} C_DIS
LIN {X 0.012,Y -553.254,Z 357.071,A 0.000,B 0.000,C 90.000,E1 48.728} C_DIS
LIN {X 0.137,Y -553.626,Z 357.066,A 0.000,B 0.000,C 90.000,E1 47.877} C_DIS
LIN {X -0.138,Y -553.710,Z 357.061,A 0.000,B 0.000,C 90.000,E1 47.067} C_DIS
LIN {X -0.355,Y -553.269,Z 357.055,A 0.000,B 0.000,C 90.000,E1 45.972} C_DIS
LIN {X 0.158,Y -552.849,Z 357.051,A 0.000,B 0.000,C 90.000,E1 45.081} C_DIS
LIN {X 0.311,Y -551.840,Z 357.044,A 0.000,B 0.000,C 90.000,E1 43.947} C_DIS
LIN {X 0.066,Y -550.612,Z 357.038,A 0.000,B 0.000,C 90.000,E1 42.852} C_DIS
LIN {X -0.195,Y -549.208,Z 357.032,A 0.000,B 0.000,C 90.000,E1 41.757} C_DIS
LIN {X 0.022,Y -546.938,Z 357.023,A 0.000,B 0.000,C 90.000,E1 40.048} C_DIS
LIN {X -0.231,Y -544.662,Z 357.013,A 0.000,B 0.000,C 90.000,E1 38.382} C_DIS
LIN {X -0.024,Y -542.440,Z 357.004,A 0.000,B 0.000,C 90.000,E1 36.664} C_DIS
LIN {X 0.130,Y -540.238,Z 356.994,A 0.000,B 0.000,C 90.000,E1 34.945} C_DIS
LIN {X 0.064,Y -538.060,Z 356.985,A 0.000,B 0.000,C 90.000,E1 33.245} C_DIS
LIN {X -0.330,Y -535.321,Z 356.972,A 0.000,B 0.000,C 90.000,E1 31.003} C_DIS
LIN {X -0.160,Y -532.742,Z 356.959,A 0.000,B 0.000,C 90.000,E1 28.693} C_DIS
LIN {X 0.015,Y -530.903,Z 356.950,A 0.000,B 0.000,C 90.000,E1 26.950} C_DIS
LIN {X 0.021,Y -528.546,Z 356.937,A 0.000,B 0.000,C 90.000,E1 24.643} C_DIS
LIN {X -0.229,Y -527.452,Z 356.931,A 0.000,B 0.000,C 90.000,E1 23.515} C_DIS
LIN {X -0.001,Y -525.478,Z 356.918,A 0.000,B 0.000,C 90.000,E1 21.173} C_DIS
LIN {X -0.160,Y -524.207,Z 356.908,A 0.000,B 0.000,C 90.000,E1 19.450} C_DIS
LIN {X -0.044,Y -523.079,Z 356.897,A 0.000,B 0.000,C 90.000,E1 17.402} C_DIS
LIN {X 0.033,Y -522.042,Z 356.882,A 0.000,B 0.000,C 90.000,E1 14.773} C_DIS
LIN {X 0.186,Y -521.633,Z 356.871,A 0.000,B 0.000,C 90.000,E1 12.715} C_DIS
LIN {X -0.266,Y -521.678,Z 356.855,A 0.000,B 0.000,C 90.000,E1 9.849} C_DIS
LIN {X 0.125,Y -522.234,Z 356.842,A 0.000,B 0.000,C 90.000,E1 7.473} C_DIS
LIN {X 0.002,Y -523.054,Z 356.832,A 0.000,B 0.000,C 90.000,E1 5.739} C_DIS
LIN {X 0.084,Y -526.035,Z 356.809,A 0.000,B 0.000,C 90.000,E1 1.661} C_DIS
LIN {X 0.081,Y -530.312,Z 356.789,A 0.000,B 0.000,C 90.000,E1 358.051} C_DIS
LIN {X -0.003,Y -533.377,Z 356.778,A 0.000,B 0.000,C 90.000,E1 356.045} C_DIS
LIN {X 0.063,Y -536.371,Z 356.769,A 0.000,B 0.000,C 90.000,E1 354.318} C_DIS
LIN {X 0.006,Y -542.984,Z 356.750,A 0.000,B 0.000,C 90.000,E1 350.905} C_DIS
LIN {X 0.255,Y -545.531,Z 356.743,A 0.000,B 0.000,C 90.000,E1 349.746} C_DIS
LIN {X -0.084,Y -554.287,Z 356.724,A 0.000,B 0.000,C 90.000,E1 346.408} C_DIS
LIN {X -0.263,Y -559.128,Z 356.715,A 0.000,B 0.000,C 90.000,E1 344.755} C_DIS
LIN {X 0.119,Y -565.079,Z 356.704,A 0.000,B 0.000,C 90.000,E1 342.779} C_DIS
LIN {X -0.081,Y -571.952,Z 356.692,A 0.000,B 0.000,C 90.000,E1 340.604} C_DIS
LIN {X 0.253,Y -576.319,Z 356.685,A 0.000,B 0.000,C 90.000,E1 339.209} C_DIS
LIN {X 0.218,Y -583.198,Z 356.673,A 0.000,B 0.000,C 90.000,E1 337.050} C_DIS
LIN {X 0.172,Y -589.312,Z 356.662,A 0.000,B 0.000,C 90.000,E1 335.177} C_DIS
LIN {X 0.174,Y -593.757,Z 356.655,A 0.000,B 0.000,C 90.000,E1 333.845} C_DIS
LIN {X 0.074,Y -597.407,Z 356.649,A 0.000,B 0.000,C 90.000,E1 332.794} C_DIS
LIN {X -0.100,Y -602.852,Z 356.640,A 0.000,B 0.000,C 90.000,E1 331.229} C_DIS
LIN {X 0.033,Y -610.212,Z 356.629,A 0.000,B 0.000,C 90.000,E1 329.125} C_DIS
LIN {X 0.165,Y -613.834,Z 356.623,A 0.000,B 0.000,C 90.000,E1 328.074} C_DIS
LIN {X -0.130,Y -620.291,Z 356.613,A 0.000,B 0.000,C 90.000,E1 326.294} C_DIS
LIN {X 0.271,Y -624.846,Z 356.606,A 0.000,B 0.000,C 90.000,E1 324.975} C_DIS
LIN {X -0.109,Y -628.456,Z 356.600,A 0.000,B 0.000,C 90.000,E1 323.989} C_DIS
LIN {X -0.068,Y -632.015,Z 356.594,A 0.000,B 0.000,C 90.000,E1 322.970} C_DIS
LIN {X -0.103,Y -637.256,Z 356.586,A 0.000,B 0.000,C 90.000,E1 321.457} C_DIS
LIN {X 0.178,Y -645.295,Z 356.573,A 0.000,B 0.000,C 90.000,E1 319.175} C_DIS
LIN {X 0.374,Y -648.648,Z 356.568,A 0.000,B 0.000,C 90.000,E1 318.162} C_DIS
LIN {X -0.048,Y -656.311,Z 356.555,A 0.000,B 0.000,C 90.000,E1 315.972} C_DIS
LIN {X -0.173,Y -659.681,Z 356.550,A 0.000,B 0.000,C 90.000,E1 315.000} C_DIS
LIN {X 0.193,Y -665.466,Z 356.540,A 0.000,B 0.000,C 90.000,E1 313.257} C_DIS
LIN {X -0.268,Y -669.587,Z 356.534,A 0.000,B 0.000,C 90.000,E1 312.081} C_DIS
LIN {X -0.168,Y -673.353,Z 356.527,A 0.000,B 0.000,C 90.000,E1 310.862} C_DIS
LIN {X 0.010,Y -677.754,Z 356.519,A 0.000,B 0.000,C 90.000,E1 309.402} C_DIS
LIN {X 0.331,Y -681.233,Z 356.512,A 0.000,B 0.000,C 90.000,E1 308.177} C_DIS
LIN {X 0.145,Y -683.803,Z 356.507,A 0.000,B 0.000,C 90.000,E1 307.237} C_DIS
LIN {X -0.013,Y -686.105,Z 356.502,A 0.000,B 0.000,C 90.000,E1 306.297} C_DIS
LIN {X -0.151,Y -688.123,Z 356.496,A 0.000,B 0.000,C 90.000,E1 305.358} C_DIS
LIN {X 0.266,Y -689.480,Z 356.492,A 0.000,B 0.000,C 90.000,E1 304.612} C_DIS
LIN {X 0.133,Y -690.728,Z 356.489,A 0.000,B 0.000,C 90.000,E1 303.913} C_DIS
LIN {X 0.228,Y -692.018,Z 356.483,A 0.000,B 0.000,C 90.000,E1 302.959} C_DIS
LIN {X 0.340,Y -692.979,Z 356.478,A 0.000,B 0.000,C 90.000,E1 302.005} C_DIS
LIN {X -0.137,Y -693.473,Z 356.474,A 0.000,B 0.000,C 90.000,E1 301.337} C_DIS
LIN {X 0.342,Y -693.626,Z 356.470,A 0.000,B 0.000,C 90.000,E1 300.590} C_DIS
LIN {X -0.132,Y -693.373,Z 356.466,A 0.000,B 0.000,C 90.000,E1 299.922} C_DIS
LIN {X -0.250,Y -693.123,Z 356.464,A 0.000,B 0.000,C 90.000,E1 299.461} C_DIS
LIN {X -0.126,Y -692.426,Z 356.460,A 0.000,B 0.000,C 90.000,E1 298.743} C_DIS
LIN {X 0.232,Y -691.091,Z 356.454,A 0.000,B 0.000,C 90.000,E1 297.769} C_DIS
LIN {X -0.123,Y -688.904,Z 356.448,A 0.000,B 0.000,C 90.000,E1 296.616} C_DIS
LIN {X -0.118,Y -687.034,Z 356.443,A 0.000,B 0.000,C 90.000,E1 295.668} C_DIS
LIN {X 0.086,Y -684.360,Z 356.436,A 0.000,B 0.000,C 90.000,E1 294.463} C_DIS
LIN {X 0.171,Y -680.961,Z 356.428,A 0.000,B 0.000,C 90.000,E1 293.025} C_DIS
LIN {X 0.181,Y -677.337,Z 356.420,A 0.000,B 0.000,C 90.000,E1 291.589} C_DIS
LIN {X -0.139,Y -673.660,Z 356.412,A 0.000,B 0.000,C 90.000,E1 290.174} C_DIS
LIN {X -0.063,Y -668.780,Z 356.401,A 0.000,B 0.000,C 90.000,E1 288.236} C_DIS
LIN {X 0.146,Y -663.122,Z 356.388,A 0.000,B 0.000,C 90.000,E1 285.788} C_DIS
LIN {X 0.000,Y -657.963,Z 356.374,A 0.000,B 0.000,C 90.000,E1 283.355} C_DIS
LIN {X -0.221,Y -652.992,Z 356.358,A 0.000,B 0.000,C 90.000,E1 280.423} C_DIS
LIN {X 0.169,Y -648.489,Z 356.336,A 0.000,B 0.000,C 90.000,E1 276.429} C_DIS
LIN {X 0.236,Y -646.988,Z 356.323,A 0.000,B 0.000,C 90.000,E1 274.188} C_DIS
LIN {X -0.191,Y -646.017,Z 356.308,A 0.000,B 0.000,C 90.000,E1 271.489} C_DIS
LIN {X -0.070,Y -646.135,Z 356.289,A 0.000,B 0.000,C 90.000,E1 267.993} C_DIS
LIN {X -0.079,Y -647.043,Z 356.276,A 0.000,B 0.000,C 90.000,E1 265.755} C_DIS
LIN {X 0.202,Y -648.008,Z 356.265,A 0.000,B 0.000,C 90.000,E1 263.742} C_DIS
LIN {X 0.165,Y -648.908,Z 356.256,A 0.000,B 0.000,C 90.000,E1 262.008} C_DIS
LIN {X -0.112,Y -649.686,Z 356.249,A 0.000,B 0.000,C 90.000,E1 260.792} C_DIS
LIN {X -0.022,Y -650.255,Z 356.239,A 0.000,B 0.000,C 90.000,E1 259.050} C_DIS
LIN {X -0.042,Y -650.759,Z 356.232,A 0.000,B 0.000,C 90.000,E1 257.813} C_DIS
LIN {X -0.065,Y -651.127,Z 356.227,A 0.000,B 0.000,C 90.000,E1 256.825} C_DIS
LIN {X 0.055,Y -651.171,Z 356.221,A 0.000,B 0.000,C 90.000,E1 255.825} C_DIS
LIN {X -0.163,Y -650.953,Z 356.217,A 0.000,B 0.000,C 90.000,E1 255.102} C_DIS
LIN {X 0.211,Y -650.713,Z 356.214,A 0.000,B 0.000,C 90.000,E1 254.574} C_DIS
LIN {X 0.081,Y -650.428,Z 356.213,A 0.000,B 0.000,C 90.000,E1 254.338} C_DIS
LIN {X -0.048,Y -650.349,Z 356.212,A 0.000,B 0.000,C 90.000,E1 254.102} C_DIS
LIN {X -0.181,Y -650.033,Z 356.210,A 0.000,B 0.000,C 90.000,E1 253.866} C_DIS
LIN {X -0.262,Y -649.634,Z 356.208,A 0.000,B 0.000,C 90.000,E1 253.378} C_DIS
LIN {X 0.090,Y -649.050,Z 356.205,A 0.000,B 0.000,C 90.000,E1 252.851} C_DIS
LIN {X -0.075,Y -647.455,Z 356.199,A 0.000,B 0.000,C 90.000,E1 251.873} C_DIS
LIN {X 0.307,Y -646.009,Z 356.195,A 0.000,B 0.000,C 90.000,E1 251.094} C_DIS
LIN {X 0.057,Y -644.234,Z 356.191,A 0.000,B 0.000,C 90.000,E1 250.369} C_DIS
LIN {X 0.011,Y -642.078,Z 356.187,A 0.000,B 0.000,C 90.000,E1 249.625} C_DIS
LIN {X 0.184,Y -638.043,Z 356.180,A 0.000,B 0.000,C 90.000,E1 248.358} C_DIS
LIN {X 0.080,Y -635.437,Z 356.176,A 0.000,B 0.000,C 90.000,E1 247.614} C_DIS
LIN {X 0.048,Y -629.723,Z 356.167,A 0.000,B 0.000,C 90.000,E1 246.102} C_DIS
LIN {X -0.116,Y -625.777,Z 356.162,A 0.000,B 0.000,C 90.000,E1 245.101} C_DIS
LIN {X -0.062,Y -620.703,Z 356.155,A 0.000,B 0.000,C 90.000,E1 243.819} C_DIS
LIN {X -0.128,Y -613.503,Z 356.145,A 0.000,B 0.000,C 90.000,E1 242.025} C_DIS
LIN {X 0.005,Y -608.360,Z 356.137,A 0.000,B 0.000,C 90.000,E1 240.717} C_DIS
LIN {X 0.217,Y -601.186,Z 356.127,A 0.000,B 0.000,C 90.000,E1 238.869} C_DIS
LIN {X 0.050,Y -594.163,Z 356.117,A 0.000,B 0.000,C 90.000,E1 237.041} C_DIS
LIN {X 0.094,Y -585.678,Z 356.104,A 0.000,B 0.000,C 90.000,E1 234.642} C_DIS
LIN {X -0.268,Y -581.270,Z 356.096,A 0.000,B 0.000,C 90.000,E1 233.336} C_DIS
LIN {X -0.040,Y -577.455,Z 356.090,A 0.000,B 0.000,C 90.000,E1 232.236} C_DIS
LIN {X -0.223,Y -573.532,Z 356.084,A 0.000,B 0.000,C 90.000,E1 231.170} C_DIS
LIN {X -0.005,Y -565.048,Z 356.071,A 0.000,B 0.000,C 90.000,E1 228.690} C_DIS
LIN {X 0.022,Y -560.544,Z 356.063,A 0.000,B 0.000,C 90.000,E1 227.310} C_DIS
LIN {X 0.004,Y -555.090,Z 356.054,A 0.000,B 0.000,C 90.000,E1 225.648} C_DIS
LIN {X 0.256,Y -549.661,Z 356.044,A 0.000,B 0.000,C 90.000,E1 223.947} C_DIS
LIN {X -0.022,Y -546.089,Z 356.038,A 0.000,B 0.000,C 90.000,E1 222.852} C_DIS
LIN {X 0.054,Y -540.769,Z 356.029,A 0.000,B 0.000,C 90.000,E1 221.148} C_DIS
LIN {X 0.071,Y -535.567,Z 356.019,A 0.000,B 0.000,C 90.000,E1 219.439} C_DIS
LIN {X -0.038,Y -529.591,Z 356.008,A 0.000,B 0.000,C 90.000,E1 217.443} C_DIS
LIN {X 0.218,Y -523.883,Z 355.997,A 0.000,B 0.000,C 90.000,E1 215.391} C_DIS
LIN {X -0.030,Y -517.733,Z 355.984,A 0.000,B 0.000,C 90.000,E1 213.086} C_DIS
LIN {X -0.235,Y -511.435,Z 355.969,A 0.000,B 0.000,C 90.000,E1 210.463} C_DIS
LIN {X 0.026,Y -506.790,Z 355.958,A 0.000,B 0.000,C 90.000,E1 208.359} C_DIS
LIN {X -0.082,Y -502.196,Z 355.946,A 0.000,B 0.000,C 90.000,E1 206.283} C_DIS
LIN {X 0.028,Y -498.962,Z 355.938,A 0.000,B 0.000,C 90.000,E1 204.771} C_DIS
LIN {X -0.236,Y -496.937,Z 355.933,A 0.000,B 0.000,C 90.000,E1 203.898} C_DIS
LIN {X -0.179,Y -492.835,Z 355.923,A 0.000,B 0.000,C 90.000,E1 202.078} C_DIS
LIN {X -0.021,Y -489.997,Z 355.916,A 0.000,B 0.000,C 90.000,E1 200.844} C_DIS
LIN {X -0.185,Y -485.125,Z 355.904,A 0.000,B 0.000,C 90.000,E1 198.725} C_DIS
LIN {X -0.167,Y -479.819,Z 355.890,A 0.000,B 0.000,C 90.000,E1 196.260} C_DIS
LIN {X 0.049,Y -475.460,Z 355.878,A 0.000,B 0.000,C 90.000,E1 194.064} C_DIS
LIN {X -0.148,Y -470.744,Z 355.864,A 0.000,B 0.000,C 90.000,E1 191.591} C_DIS
LIN {X -0.033,Y -466.675,Z 355.852,A 0.000,B 0.000,C 90.000,E1 189.378} C_DIS
LIN {X 0.037,Y -463.544,Z 355.842,A 0.000,B 0.000,C 90.000,E1 187.473} C_DIS
LIN {X -0.213,Y -459.156,Z 355.826,A 0.000,B 0.000,C 90.000,E1 184.645} C_DIS
LIN {X -0.192,Y -454.500,Z 355.804,A 0.000,B 0.000,C 90.000,E1 180.802} C_DIS
LIN {X -0.102,Y -451.526,Z 355.785,A 0.000,B 0.000,C 90.000,E1 177.249} C_DIS
LIN {X 0.161,Y -449.800,Z 355.763,A 0.000,B 0.000,C 90.000,E1 173.337} C_DIS
LIN {X 0.139,Y -449.661,Z 355.742,A 0.000,B 0.000,C 90.000,E1 169.454} C_DIS
LIN {X -0.234,Y -450.544,Z 355.725,A 0.000,B 0.000,C 90.000,E1 166.589} C_DIS
LIN {X 0.114,Y -453.176,Z 355.704,A 0.000,B 0.000,C 90.000,E1 162.670} C_DIS
LIN {X -0.030,Y -455.763,Z 355.690,A 0.000,B 0.000,C 90.000,E1 160.115} C_DIS
LIN {X 0.080,Y -459.120,Z 355.675,A 0.000,B 0.000,C 90.000,E1 157.539} C_DIS
LIN {X 0.069,Y -464.188,Z 355.658,A 0.000,B 0.000,C 90.000,E1 154.357} C_DIS
LIN {X 0.100,Y -472.677,Z 355.635,A 0.000,B 0.000,C 90.000,E1 150.255} C_DIS
LIN {X -0.123,Y -482.580,Z 355.614,A 0.000,B 0.000,C 90.000,E1 146.548} C_DIS
LIN {X 0.060,Y -490.226,Z 355.600,A 0.000,B 0.000,C 90.000,E1 144.069} C_DIS
LIN {X -0.166,Y -496.282,Z 355.590,A 0.000,B 0.000,C 90.000,E1 142.271} C_DIS
LIN {X 0.176,Y -501.303,Z 355.582,A 0.000,B 0.000,C 90.000,E1 140.723} C_DIS
LIN {X 0.016,Y -505.127,Z 355.575,A 0.000,B 0.000,C 90.000,E1 139.542} C_DIS
LIN {X 0.239,Y -508.740,Z 355.569,A 0.000,B 0.000,C 90.000,E1 138.324} C_DIS
LIN {X 0.140,Y -512.190,Z 355.562,A 0.000,B 0.000,C 90.000,E1 137.148} C_DIS
LIN {X -0.172,Y -514.419,Z 355.557,A 0.000,B 0.000,C 90.000,E1 136.296} C_DIS
LIN {X -0.104,Y -516.432,Z 355.552,A 0.000,B 0.000,C 90.000,E1 135.405} C_DIS
LIN {X -0.289,Y -517.700,Z 355.549,A 0.000,B 0.000,C 90.000,E1 134.838} C_DIS
LIN {X -0.185,Y -519.238,Z 355.544,A 0.000,B 0.000,C 90.000,E1 133.947} C_DIS
LIN {X -0.066,Y -520.399,Z 355.539,A 0.000,B 0.000,C 90.000,E1 133.056} C_DIS
LIN {X -0.006,Y -521.377,Z 355.533,A 0.000,B 0.000,C 90.000,E1 131.881} C_DIS
LIN {X 0.168,Y -521.796,Z 355.528,A 0.000,B 0.000,C 90.000,E1 130.987} C_DIS
LIN {X -0.048,Y -521.793,Z 355.523,A 0.000,B 0.000,C 90.000,E1 130.135} C_DIS
LIN {X -0.149,Y -521.668,Z 355.520,A 0.000,B 0.000,C 90.000,E1 129.564} C_DIS
LIN {X 0.033,Y -521.143,Z 355.515,A 0.000,B 0.000,C 90.000,E1 128.669} C_DIS
LIN {X -0.166,Y -519.907,Z 355.508,A 0.000,B 0.000,C 90.000,E1 127.523} C_DIS
LIN {X 0.289,Y -518.023,Z 355.500,A 0.000,B 0.000,C 90.000,E1 126.011} C_DIS
LIN {X -0.320,Y -515.883,Z 355.492,A 0.000,B 0.000,C 90.000,E1 124.612} C_DIS
LIN {X 0.249,Y -513.739,Z 355.486,A 0.000,B 0.000,C 90.000,E1 123.372} C_DIS
LIN {X 0.074,Y -511.407,Z 355.479,A 0.000,B 0.000,C 90.000,E1 122.212} C_DIS
LIN {X -0.139,Y -508.732,Z 355.472,A 0.000,B 0.000,C 90.000,E1 121.052} C_DIS
LIN {X -0.217,Y -505.959,Z 355.466,A 0.000,B 0.000,C 90.000,E1 119.873} C_DIS
LIN {X 0.046,Y -503.681,Z 355.461,A 0.000,B 0.000,C 90.000,E1 118.949} C_DIS
LIN {X -0.104,Y -500.467,Z 355.454,A 0.000,B 0.000,C 90.000,E1 117.769} C_DIS
LIN {X -0.142,Y -497.980,Z 355.449,A 0.000,B 0.000,C 90.000,E1 116.873} C_DIS
LIN {X -0.157,Y -494.468,Z 355.443,A 0.000,B 0.000,C 90.000,E1 115.668} C_DIS
LIN {X -0.261,Y -491.684,Z 355.438,A 0.000,B 0.000,C 90.000,E1 114.771} C_DIS
LIN {X 0.096,Y -486.549,Z 355.429,A 0.000,B 0.000,C 90.000,E1 113.206} C_DIS
LIN {X 0.160,Y -482.236,Z 355.422,A 0.000,B 0.000,C 90.000,E1 111.972} C_DIS
LIN {X 0.145,Y -476.268,Z 355.414,A 0.000,B 0.000,C 90.000,E1 110.429} C_DIS
LIN {X 0.081,Y -470.443,Z 355.406,A 0.000,B 0.000,C 90.000,E1 109.033} C_DIS
LIN {X -0.083,Y -464.366,Z 355.398,A 0.000,B 0.000,C 90.000,E1 107.638} C_DIS
LIN {X 0.134,Y -462.412,Z 355.396,A 0.000,B 0.000,C 90.000,E1 107.166} C_DIS
LIN {X 0.093,Y -462.416,Z 355.395,A 0.000,B 0.000,C 90.000,E1 107.166} C_DIS
LIN {X 0.237,Y -467.289,Z 355.384,A 0.000,B 0.000,C 90.000,E1 105.064} C_DIS
LIN {X 0.040,Y -467.973,Z 355.382,A 0.000,B 0.000,C 90.000,E1 104.773} C_DIS
LIN {X 0.004,Y -476.192,Z 355.356,A 0.000,B 0.000,C 90.000,E1 100.074} C_DIS
LIN {X 0.259,Y -482.096,Z 355.330,A 0.000,B 0.000,C 90.000,E1 95.391} C_DIS
LIN {X 0.009,Y -485.510,Z 355.305,A 0.000,B 0.000,C 90.000,E1 90.802} C_DIS
LIN {X 0.041,Y -486.382,Z 355.281,A 0.000,B 0.000,C 90.000,E1 86.502} C_DIS
LIN {X -0.134,Y -486.361,Z 355.279,A 0.000,B 0.000,C 90.000,E1 86.216} C_DIS
LIN {X -0.050,Y -484.682,Z 355.253,A 0.000,B 0.000,C 90.000,E1 81.602} C_DIS
LIN {X -0.150,Y -480.603,Z 355.228,A 0.000,B 0.000,C 90.000,E1 76.992} C_DIS
LIN {X 0.175,Y -480.232,Z 355.226,A 0.000,B 0.000,C 90.000,E1 76.645} C_DIS
LIN {X 0.101,Y -476.449,Z 355.212,A 0.000,B 0.000,C 90.000,E1 74.102} C_DIS
LIN {X 0.060,Y -476.467,Z 355.212,A 0.000,B 0.000,C 90.000,E1 74.102} C_DIS
LIN {X 0.273,Y -480.433,Z 355.208,A 0.000,B 0.000,C 90.000,E1 73.378} C_DIS
LIN {X -0.042,Y -485.495,Z 355.203,A 0.000,B 0.000,C 90.000,E1 72.489} C_DIS
LIN {X 0.060,Y -489.517,Z 355.198,A 0.000,B 0.000,C 90.000,E1 71.710} C_DIS
LIN {X -0.095,Y -494.413,Z 355.193,A 0.000,B 0.000,C 90.000,E1 70.678} C_DIS
LIN {X -0.005,Y -497.131,Z 355.189,A 0.000,B 0.000,C 90.000,E1 70.061} C_DIS
LIN {X -0.203,Y -501.406,Z 355.183,A 0.000,B 0.000,C 90.000,E1 69.028} C_DIS
LIN {X -0.131,Y -502.450,Z 355.182,A 0.000,B 0.000,C 90.000,E1 68.720} C_DIS
LIN {X -0.010,Y -503.686,Z 355.180,A 0.000,B 0.000,C 90.000,E1 68.411} C_DIS
LIN {X 0.152,Y -505.760,Z 355.177,A 0.000,B 0.000,C 90.000,E1 67.794} C_DIS
LIN {X 0.058,Y -509.732,Z 355.170,A 0.000,B 0.000,C 90.000,E1 66.613} C_DIS
LIN {X 0.230,Y -513.397,Z 355.164,A 0.000,B 0.000,C 90.000,E1 65.409} C_DIS
LIN {X -0.225,Y -516.875,Z 355.157,A 0.000,B 0.000,C 90.000,E1 64.280} C_DIS
LIN {X 0.095,Y -521.936,Z 355.147,A 0.000,B 0.000,C 90.000,E1 62.487} C_DIS
LIN {X -0.089,Y -525.969,Z 355.139,A 0.000,B 0.000,C 90.000,E1 61.051} C_DIS
LIN {X -0.242,Y -530.775,Z 355.130,A 0.000,B 0.000,C 90.000,E1 59.331} C_DIS
LIN {X -0.016,Y -535.511,Z 355.120,A 0.000,B 0.000,C 90.000,E1 57.582} C_DIS
LIN {X 0.138,Y -538.568,Z 355.114,A 0.000,B 0.000,C 90.000,E1 56.421} C_DIS
LIN {X -0.091,Y -542.170,Z 355.106,A 0.000,B 0.000,C 90.000,E1 55.022} C_DIS
LIN {X -0.324,Y -544.177,Z 355.101,A 0.000,B 0.000,C 90.000,E1 54.196} C_DIS
LIN {X -0.180,Y -546.688,Z 355.095,A 0.000,B 0.000,C 90.000,E1 53.050} C_DIS
LIN {X -0.048,Y -548.434,Z 355.090,A 0.000,B 0.000,C 90.000,E1 52.190} C_DIS
LIN {X -0.276,Y -550.452,Z 355.084,A 0.000,B 0.000,C 90.000,E1 51.090} C_DIS
LIN {X -0.113,Y -551.690,Z 355.079,A 0.000,B 0.000,C 90.000,E1 50.231} C_DIS
LIN {X -0.308,Y -553.211,Z 355.071,A 0.000,B 0.000,C 90.000,E1 48.852} C_DIS
LIN {X -0.179,Y -553.738,Z 355.067,A 0.000,B 0.000,C 90.000,E1 48.000} C_DIS
LIN {X 0.012,Y -554.032,Z 355.060,A 0.000,B 0.000,C 90.000,E1 46.863} C_DIS
LIN {X 0.179,Y -553.686,Z 355.054,A 0.000,B 0.000,C 90.000,E1 45.729} C_DIS
LIN {X 0.264,Y -553.465,Z 355.051,A 0.000,B 0.000,C 90.000,E1 45.162} C_DIS
LIN {X -0.355,Y -552.570,Z 355.045,A 0.000,B 0.000,C 90.000,E1 44.109} C_DIS
LIN {X 0.145,Y -551.741,Z 355.040,A 0.000,B 0.000,C 90.000,E1 43.218} C_DIS
LIN {X 0.256,Y -550.802,Z 355.036,A 0.000,B 0.000,C 90.000,E1 42.366} C_DIS
LIN {X -0.007,Y -549.738,Z 355.031,A 0.000,B 0.000,C 90.000,E1 41.553} C_DIS
LIN {X -0.239,Y -547.929,Z 355.023,A 0.000,B 0.000,C 90.000,E1 40.172} C_DIS
LIN {X -0.049,Y -545.661,Z 355.014,A 0.000,B 0.000,C 90.000,E1 38.463} C_DIS
LIN {X -0.221,Y -543.057,Z 355.003,A 0.000,B 0.000,C 90.000,E1 36.503} C_DIS
LIN {X 0.098,Y -540.497,Z 354.992,A 0.000,B 0.000,C 90.000,E1 34.485} C_DIS
LIN {X -0.112,Y -538.322,Z 354.982,A 0.000,B 0.000,C 90.000,E1 32.801} C_DIS
LIN {X -0.042,Y -536.303,Z 354.973,A 0.000,B 0.000,C 90.000,E1 31.082} C_DIS
LIN {X 0.264,Y -534.346,Z 354.963,A 0.000,B 0.000,C 90.000,E1 29.333} C_DIS
LIN {X -0.006,Y -532.553,Z 354.954,A 0.000,B 0.000,C 90.000,E1 27.641} C_DIS
LIN {X -0.079,Y -530.708,Z 354.944,A 0.000,B 0.000,C 90.000,E1 25.924} C_DIS
LIN {X -0.004,Y -528.776,Z 354.933,A 0.000,B 0.000,C 90.000,E1 23.898} C_DIS
LIN {X -0.026,Y -526.765,Z 354.920,A 0.000,B 0.000,C 90.000,E1 21.589} C_DIS
LIN {X -0.175,Y -525.270,Z 354.909,A 0.000,B 0.000,C 90.000,E1 19.577} C_DIS
LIN {X 0.131,Y -524.122,Z 354.897,A 0.000,B 0.000,C 90.000,E1 17.511} C_DIS
LIN {X 0.095,Y -523.073,Z 354.883,A 0.000,B 0.000,C 90.000,E1 14.898} C_DIS
LIN {X -0.110,Y -522.642,Z 354.872,A 0.000,B 0.000,C 90.000,E1 12.883} C_DIS
LIN {X -0.027,Y -522.675,Z 354.855,A 0.000,B 0.000,C 90.000,E1 9.962} C_DIS
LIN {X -0.128,Y -523.340,Z 354.841,A 0.000,B 0.000,C 90.000,E1 7.352} C_DIS
LIN {X 0.232,Y -524.182,Z 354.831,A 0.000,B 0.000,C 90.000,E1 5.568} C_DIS
LIN {X -0.101,Y -526.674,Z 354.812,A 0.000,B 0.000,C 90.000,E1 2.121} C_DIS
LIN {X 0.104,Y -531.055,Z 354.791,A 0.000,B 0.000,C 90.000,E1 358.339} C_DIS
LIN {X 0.079,Y -534.927,Z 354.777,A 0.000,B 0.000,C 90.000,E1 355.755} C_DIS
LIN {X 0.133,Y -537.929,Z 354.767,A 0.000,B 0.000,C 90.000,E1 354.033} C_DIS
LIN {X 0.126,Y -544.634,Z 354.748,A 0.000,B 0.000,C 90.000,E1 350.622} C_DIS
LIN {X 0.151,Y -548.540,Z 354.739,A 0.000,B 0.000,C 90.000,E1 348.926} C_DIS
LIN {X 0.224,Y -556.080,Z 354.723,A 0.000,B 0.000,C 90.000,E1 346.117} C_DIS
LIN {X 0.232,Y -560.947,Z 354.714,A 0.000,B 0.000,C 90.000,E1 344.448} C_DIS
LIN {X -0.034,Y -566.941,Z 354.703,A 0.000,B 0.000,C 90.000,E1 342.543} C_DIS
LIN {X -0.167,Y -572.108,Z 354.694,A 0.000,B 0.000,C 90.000,E1 340.913} C_DIS
LIN {X 0.001,Y -577.371,Z 354.685,A 0.000,B 0.000,C 90.000,E1 339.263} C_DIS
LIN {X 0.001,Y -584.269,Z 354.673,A 0.000,B 0.000,C 90.000,E1 337.102} C_DIS
LIN {X -0.121,Y -591.300,Z 354.661,A 0.000,B 0.000,C 90.000,E1 334.973} C_DIS
LIN {X -0.257,Y -597.636,Z 354.651,A 0.000,B 0.000,C 90.000,E1 333.127} C_DIS
LIN {X 0.025,Y -603.975,Z 354.640,A 0.000,B 0.000,C 90.000,E1 331.257} C_DIS
LIN {X 0.221,Y -610.414,Z 354.630,A 0.000,B 0.000,C 90.000,E1 329.410} C_DIS
LIN {X 0.114,Y -615.046,Z 354.623,A 0.000,B 0.000,C 90.000,E1 328.122} C_DIS
LIN {X 0.060,Y -620.515,Z 354.614,A 0.000,B 0.000,C 90.000,E1 326.580} C_DIS
LIN {X 0.155,Y -623.264,Z 354.610,A 0.000,B 0.000,C 90.000,E1 325.801} C_DIS
LIN {X 0.268,Y -626.822,Z 354.604,A 0.000,B 0.000,C 90.000,E1 324.769} C_DIS
LIN {X -0.089,Y -630.335,Z 354.599,A 0.000,B 0.000,C 90.000,E1 323.783} C_DIS
LIN {X 0.112,Y -632.973,Z 354.595,A 0.000,B 0.000,C 90.000,E1 323.004} C_DIS
LIN {X 0.096,Y -637.212,Z 354.588,A 0.000,B 0.000,C 90.000,E1 321.743} C_DIS
LIN {X 0.382,Y -644.951,Z 354.575,A 0.000,B 0.000,C 90.000,E1 319.461} C_DIS
LIN {X -0.269,Y -647.529,Z 354.571,A 0.000,B 0.000,C 90.000,E1 318.771} C_DIS
LIN {X -0.208,Y -654.138,Z 354.560,A 0.000,B 0.000,C 90.000,E1 316.782} C_DIS
LIN {X 0.072,Y -658.433,Z 354.553,A 0.000,B 0.000,C 90.000,E1 315.526} C_DIS
LIN {X -0.051,Y -662.489,Z 354.546,A 0.000,B 0.000,C 90.000,E1 314.312} C_DIS
LIN {X -0.086,Y -666.604,Z 354.539,A 0.000,B 0.000,C 90.000,E1 313.095} C_DIS
LIN {X 0.415,Y -670.668,Z 354.533,A 0.000,B 0.000,C 90.000,E1 311.838} C_DIS
LIN {X 0.009,Y -673.668,Z 354.527,A 0.000,B 0.000,C 90.000,E1 310.906} C_DIS
LIN {X -0.246,Y -678.070,Z 354.519,A 0.000,B 0.000,C 90.000,E1 309.483} C_DIS
LIN {X -0.057,Y -680.861,Z 354.514,A 0.000,B 0.000,C 90.000,E1 308.508} C_DIS
LIN {X 0.285,Y -683.496,Z 354.509,A 0.000,B 0.000,C 90.000,E1 307.523} C_DIS
LIN {X 0.093,Y -685.284,Z 354.505,A 0.000,B 0.000,C 90.000,E1 306.824} C_DIS
LIN {X 0.331,Y -686.886,Z 354.501,A 0.000,B 0.000,C 90.000,E1 306.091} C_DIS
LIN {X -0.192,Y -688.787,Z 354.495,A 0.000,B 0.000,C 90.000,E1 305.185} C_DIS
LIN {X 0.267,Y -690.398,Z 354.490,A 0.000,B 0.000,C 90.000,E1 304.199} C_DIS
LIN {X -0.456,Y -691.118,Z 354.488,A 0.000,B 0.000,C 90.000,E1 303.785} C_DIS
LIN {X 0.004,Y -691.987,Z 354.484,A 0.000,B 0.000,C 90.000,E1 303.038} C_DIS
LIN {X 0.119,Y -692.786,Z 354.478,A 0.000,B 0.000,C 90.000,E1 302.084} C_DIS
LIN {X 0.239,Y -693.237,Z 354.473,A 0.000,B 0.000,C 90.000,E1 301.131} C_DIS
LIN {X 0.122,Y -693.233,Z 354.470,A 0.000,B 0.000,C 90.000,E1 300.669} C_DIS
LIN {X 0.006,Y -693.067,Z 354.468,A 0.000,B 0.000,C 90.000,E1 300.207} C_DIS
LIN {X 0.133,Y -692.575,Z 354.464,A 0.000,B 0.000,C 90.000,E1 299.489} C_DIS
LIN {X -0.349,Y -691.840,Z 354.460,A 0.000,B 0.000,C 90.000,E1 298.821} C_DIS
LIN {X 0.005,Y -690.398,Z 354.455,A 0.000,B 0.000,C 90.000,E1 297.847} C_DIS
LIN {X 0.339,Y -688.642,Z 354.449,A 0.000,B 0.000,C 90.000,E1 296.873} C_DIS
LIN {X -0.053,Y -686.281,Z 354.443,A 0.000,B 0.000,C 90.000,E1 295.720} C_DIS
LIN {X 0.132,Y -683.564,Z 354.436,A 0.000,B 0.000,C 90.000,E1 294.515} C_DIS
LIN {X 0.194,Y -680.134,Z 354.428,A 0.000,B 0.000,C 90.000,E1 293.078} C_DIS
LIN {X -0.067,Y -676.461,Z 354.420,A 0.000,B 0.000,C 90.000,E1 291.663} C_DIS
LIN {X -0.393,Y -672.758,Z 354.412,A 0.000,B 0.000,C 90.000,E1 290.248} C_DIS
LIN {X -0.197,Y -667.242,Z 354.400,A 0.000,B 0.000,C 90.000,E1 288.055} C_DIS
LIN {X 0.054,Y -662.163,Z 354.388,A 0.000,B 0.000,C 90.000,E1 285.843} C_DIS
LIN {X -0.129,Y -656.977,Z 354.374,A 0.000,B 0.000,C 90.000,E1 283.411} C_DIS
LIN {X 0.129,Y -652.007,Z 354.358,A 0.000,B 0.000,C 90.000,E1 280.433} C_DIS
LIN {X -0.062,Y -647.474,Z 354.336,A 0.000,B 0.000,C 90.000,E1 276.486} C_DIS
LIN {X -0.211,Y -645.824,Z 354.322,A 0.000,B 0.000,C 90.000,E1 274.012} C_DIS
LIN {X 0.152,Y -644.984,Z 354.308,A 0.000,B 0.000,C 90.000,E1 271.489} C_DIS
LIN {X 0.226,Y -645.088,Z 354.289,A 0.000,B 0.000,C 90.000,E1 267.993} C_DIS
LIN {X 0.186,Y -645.998,Z 354.277,A 0.000,B 0.000,C 90.000,E1 265.755} C_DIS
LIN {X -0.203,Y -646.988,Z 354.266,A 0.000,B 0.000,C 90.000,E1 263.799} C_DIS
LIN {X -0.263,Y -647.904,Z 354.256,A 0.000,B 0.000,C 90.000,E1 262.064} C_DIS
LIN {X 0.087,Y -648.716,Z 354.249,A 0.000,B 0.000,C 90.000,E1 260.792} C_DIS
LIN {X 0.156,Y -649.410,Z 354.239,A 0.000,B 0.000,C 90.000,E1 259.050} C_DIS
LIN {X -0.015,Y -650.018,Z 354.232,A 0.000,B 0.000,C 90.000,E1 257.825} C_DIS
LIN {X 0.090,Y -650.550,Z 354.227,A 0.000,B 0.000,C 90.000,E1 256.825} C_DIS
LIN {X -0.170,Y -650.740,Z 354.224,A 0.000,B 0.000,C 90.000,E1 256.353} C_DIS
LIN {X -0.299,Y -650.701,Z 354.223,A 0.000,B 0.000,C 90.000,E1 256.117} C_DIS
LIN {X 0.202,Y -650.828,Z 354.221,A 0.000,B 0.000,C 90.000,E1 255.825} C_DIS
LIN {X -0.019,Y -650.756,Z 354.217,A 0.000,B 0.000,C 90.000,E1 255.102} C_DIS
LIN {X -0.274,Y -650.639,Z 354.215,A 0.000,B 0.000,C 90.000,E1 254.629} C_DIS
LIN {X 0.012,Y -650.120,Z 354.209,A 0.000,B 0.000,C 90.000,E1 253.614} C_DIS
LIN {X 0.235,Y -649.397,Z 354.205,A 0.000,B 0.000,C 90.000,E1 252.851} C_DIS
LIN {X 0.015,Y -648.307,Z 354.201,A 0.000,B 0.000,C 90.000,E1 252.127} C_DIS
LIN {X -0.212,Y -646.990,Z 354.197,A 0.000,B 0.000,C 90.000,E1 251.402} C_DIS
LIN {X -0.300,Y -646.029,Z 354.194,A 0.000,B 0.000,C 90.000,E1 250.913} C_DIS
LIN {X 0.057,Y -644.259,Z 354.190,A 0.000,B 0.000,C 90.000,E1 250.134} C_DIS
LIN {X 0.008,Y -642.192,Z 354.186,A 0.000,B 0.000,C 90.000,E1 249.390} C_DIS
LIN {X -0.233,Y -639.040,Z 354.180,A 0.000,B 0.000,C 90.000,E1 248.411} C_DIS
LIN {X -0.323,Y -636.569,Z 354.176,A 0.000,B 0.000,C 90.000,E1 247.667} C_DIS
LIN {X 0.186,Y -632.821,Z 354.170,A 0.000,B 0.000,C 90.000,E1 246.613} C_DIS
LIN {X 0.058,Y -629.076,Z 354.165,A 0.000,B 0.000,C 90.000,E1 245.613} C_DIS
LIN {X 0.146,Y -625.150,Z 354.159,A 0.000,B 0.000,C 90.000,E1 244.588} C_DIS
LIN {X -0.088,Y -620.060,Z 354.152,A 0.000,B 0.000,C 90.000,E1 243.332} C_DIS
LIN {X 0.127,Y -613.975,Z 354.143,A 0.000,B 0.000,C 90.000,E1 241.769} C_DIS
LIN {X 0.265,Y -608.857,Z 354.136,A 0.000,B 0.000,C 90.000,E1 240.461} C_DIS
